(* IEC 61131-3 sources: std_i2980_v2.06_cp053/Source/IMM/ieccontrol/GlobalBaseArchives (part 14) *)

(* ---- ABMotorLockList.pu ---- *)
IMPORT_OVER_LISTFILE
 SET_ALARM
, tsListStructMotorLock
, tsDeviceId
, FBDebugTrace
, tsTraceLevel
, tsElementMotorLock
, tsSearchDataMotorLock

END_IMPORT

ALGORITHM_BLOCK ABMotorLockList #DUMMY_EDIT_BLOCK

SYSTEM_VAR
 sv_DeviceId : tsDeviceId;
 sv_TraceLevel : tsTraceLevel;
END_VAR

SYSTEM_OBJECT
 erListOverflow : ALARM;
END_OBJECT

VAR
 mListStruct : tsListStructMotorLock;
 miNextFree : DINT;
 miLowBound : DINT;
 miHighBound : DINT;
 mbInit : BOOL;
 miLastFound : DINT;
 miActElement : DINT;
 fbDebugTrace : FBDebugTrace;
END_VAR

ALGORITHM aInit

#BEGIN_EDIT_BLOCK
miLowBound := GET_LOW_BOUND(mListStruct.List);
miHighBound := GET_HIGH_BOUND(mListStruct.List);
miNextFree := miLowBound;
miLastFound := miLowBound;
miActElement := miLowBound;
mbInit := TRUE;

;#END_EDIT_BLOCK END_ALGORITHM

ALGORITHM aAdd

VAR_INPUT
 Element : tsElementMotorLock;
END_VAR
#BEGIN_EDIT_BLOCK
IF NOT mbInit THEN RETURN;; END_IF;

IF miNextFree < miHighBound THEN

    mListStruct.List[miNextFree] := Element;
    mListStruct.Used[miNextFree] := TRUE;
    miNextFree := miNextFree + 1;
ELSE
    //error: List Full
    SET_ALARM(Name := erListOverflow,
              SubID1 := sv_DeviceId.CompId,
              SubID2 := sv_DeviceId.IndexId,
              Param1 := 'ABMotorLockList.aAdd');
END_IF;

;#END_EDIT_BLOCK END_ALGORITHM

ALGORITHM aAddAt

VAR_INPUT
 Element : tsElementMotorLock;
 iPos : DINT;
END_VAR

VAR_TEMP
 i : DINT;
END_VAR

VAR
 iStart : DINT;
 iEnd : DINT;
END_VAR
#BEGIN_EDIT_BLOCK
IF NOT mbInit THEN RETURN; END_IF;

IF miNextFree <= miHighBound THEN
    IF iPos < miHighBound AND iPos >= miLowBound THEN

        IF iPos < miNextFree THEN

            iStart := miNextFree;
            iEnd := iPos+1;
        ELSE
            i := iPos;
            iEnd := miNextFree;
        END_IF;
        miNextFree := i + 1;

        //reorganize list
        FOR i := iStart TO iEnd BY -1 DO
            mListStruct.List[i] := mListStruct.List[i-1];
            mListStruct.Used[i] := TRUE;
        END_FOR;
        //adding Element
        mListStruct.List[iPos] := Element;
        mListStruct.Used[iPos] := TRUE;
    ELSE
        //error: out of bounds
        IF sv_TraceLevel.bApplication THEN
            fbDebugTrace(sText := 'ABMotorLockList.aAddAt: Error: Out of ListBounds');
        END_IF;
    END_IF;
ELSE
    //error: List Full
    SET_ALARM(Name := erListOverflow,
            SubID1 := sv_DeviceId.CompId,
            SubID2 := sv_DeviceId.IndexId,
            Param1 := 'ABMotorLockList.aAddAt');
END_IF;

;#END_EDIT_BLOCK END_ALGORITHM

ALGORITHM aSearch

VAR_INPUT
 SearchData : tsSearchDataMotorLock;
END_VAR

VAR_OUTPUT
 Element : tsElementMotorLock;
 iPos : DINT;
 bFound : BOOL;
END_VAR

VAR_TEMP
 i : DINT;
END_VAR
#BEGIN_EDIT_BLOCK
IF NOT mbInit THEN RETURN;; END_IF;

iPos := 0;
bFound := FALSE;

FOR i := miLowBound TO miNextFree-1 DO

    IF mListStruct.List[i].SearchData = SearchData THEN

       Element := mListStruct.List[i];
       //remember foundposition for aSearchNext
       miLastFound := i;
       iPos := i;
       bFound := TRUE;
       RETURN;;
    END_IF;
END_FOR;

;#END_EDIT_BLOCK END_ALGORITHM

ALGORITHM aSearchNext

VAR_INPUT
 SearchData : tsSearchDataMotorLock;
END_VAR

VAR_OUTPUT
 Element : tsElementMotorLock;
 iPos : DINT;
 bFound : BOOL;
END_VAR

VAR_TEMP
 i : DINT;
END_VAR
#BEGIN_EDIT_BLOCK
IF NOT mbInit THEN RETURN;; END_IF;

iPos := 0;
bFound := FALSE;

FOR i := miLastFound+1 TO miNextFree-1 DO

    IF mListStruct.List[i].SearchData = SearchData THEN

       Element := mListStruct.List[i];
       //remember foundposition for then next aSearchNext
       miLastFound := i;
       iPos := i;
       bFound := TRUE;
       RETURN;;
    END_IF;
END_FOR;

;#END_EDIT_BLOCK END_ALGORITHM

ALGORITHM aRemove

VAR_INPUT
 SearchData : tsSearchDataMotorLock;
END_VAR

VAR_OUTPUT
 Element : tsElementMotorLock;
 iPos : DINT;
 bFound : BOOL;
END_VAR

VAR_TEMP
 i : DINT;
END_VAR
#BEGIN_EDIT_BLOCK
IF NOT mbInit THEN RETURN; END_IF;

iPos := 0;
bFound := FALSE;

FOR i := miLowBound TO miNextFree-1 DO

    IF mListStruct.List[i].SearchData = SearchData THEN

       iPos := i;
       bFound := TRUE;
       Element := mListStruct.List[i];
       //reorganize list
       FOR i := iPos TO miNextFree-1 DO
           mListStruct.List[i] := mListStruct.List[i+1];
       END_FOR;
       mListStruct.Used[miNextFree - 1] := FALSE;
       miNextFree := miNextFree - 1;
       RETURN;
    END_IF;
END_FOR;

;#END_EDIT_BLOCK END_ALGORITHM

ALGORITHM aRemoveAt

VAR_INPUT
 iPos : DINT;
END_VAR

VAR_OUTPUT
 Element : tsElementMotorLock;
END_VAR

VAR_TEMP
 i : DINT;
END_VAR
#BEGIN_EDIT_BLOCK
IF NOT mbInit THEN RETURN; END_IF;

IF iPos <= miHighBound AND iPos >= miLowBound THEN

    Element:= mListStruct.List[iPos];
    miActElement := iPos;

    //reorganize list
    FOR i := iPos TO miNextFree-1 DO
        mListStruct.List[i] := mListStruct.List[i+1];
    END_FOR;
    mListStruct.Used[miNextFree - 1] := FALSE;

    miNextFree := miNextFree - 1;
ELSE
    //error: out of bounds
    IF sv_TraceLevel.bApplication THEN
        fbDebugTrace(sText := 'ABMotorLockList.aRemoveAt: Error: Out of ListBounds');
    END_IF;
END_IF;

;#END_EDIT_BLOCK END_ALGORITHM

ALGORITHM aRemoveAll

VAR_TEMP
 i : DINT;
END_VAR
#BEGIN_EDIT_BLOCK
IF NOT mbInit THEN RETURN; END_IF;
FOR i := miNextFree-1 TO miLowBound DO
    //clearing the whole list
    mListStruct.Used[i] := FALSE;
END_FOR;
miNextFree := miLowBound;

;#END_EDIT_BLOCK END_ALGORITHM

ALGORITHM aElementAt

VAR_OUTPUT
 Element : tsElementMotorLock;
END_VAR

VAR_INPUT
 iPos : DINT;
END_VAR
#BEGIN_EDIT_BLOCK
IF NOT mbInit THEN RETURN; END_IF;

IF iPos <= miHighBound AND iPos >= miLowBound THEN

    Element := mListStruct.List[iPos];
    miActElement := iPos;
ELSE
    //error: out of bounds
    IF sv_TraceLevel.bApplication THEN
        fbDebugTrace(sText := 'ABMotorLockList.aElementAt: Error: Out of ListBounds');
    END_IF;
END_IF;

;#END_EDIT_BLOCK END_ALGORITHM

ALGORITHM aModifyAt

VAR_INPUT
 iPos : DINT;
END_VAR

VAR_IN_OUT
 Element : tsElementMotorLock;
END_VAR
#BEGIN_EDIT_BLOCK
IF NOT mbInit THEN RETURN; END_IF;

IF iPos <= miHighBound AND iPos >= miLowBound THEN

     mListStruct.List[iPos] := Element;
     miActElement := iPos;
ELSE
    //error: out of bounds
    IF sv_TraceLevel.bApplication THEN
        fbDebugTrace(sText := 'ABMotorLockList.aModifyAt: Error: Out of ListBounds');
    END_IF;
END_IF;

;#END_EDIT_BLOCK END_ALGORITHM

// ALGORITHM aGetSize

// #BEGIN_EDIT_BLOCK
// IF NOT mbInit THEN RETURN; END_IF;
// //returns the size of the list
// iSize := miHighBound - miLowBound;

// ;#END_EDIT_BLOCK END_ALGORITHM

// ALGORITHM aGetElementsCount

// VAR_OUTPUT
 // iUsed : DINT;
// END_VAR
// #BEGIN_EDIT_BLOCK
// IF NOT mbInit THEN RETURN; END_IF;
//
// iUsed := miNextFree - miLowBound;

// ;#END_EDIT_BLOCK END_ALGORITHM

FUNCTION aGetSize : DINT
 #DUMMY_EDIT_BLOCK
#BEGIN_EDIT_BLOCK
IF NOT mbInit THEN RETURN; END_IF;
//returns the size of the list
aGetSize := miHighBound - miLowBound;

;#END_EDIT_BLOCK END_FUNCTION

FUNCTION aGetElementCount : DINT
 #DUMMY_EDIT_BLOCK
#BEGIN_EDIT_BLOCK
IF NOT mbInit THEN RETURN; END_IF;

aGetElementCount:= miNextFree - miLowBound;

;#END_EDIT_BLOCK END_FUNCTION

ALGORITHM aFirstElement

VAR_OUTPUT
 Element : tsElementMotorLock;
END_VAR
#BEGIN_EDIT_BLOCK
IF NOT mbInit THEN RETURN; END_IF;

miActElement := miLowBound;
Element := mListStruct.List[miLowBound];

;#END_EDIT_BLOCK END_ALGORITHM

ALGORITHM aNextElement

VAR_OUTPUT
 Element : tsElementMotorLock;
 iPos : DINT;
END_VAR
#BEGIN_EDIT_BLOCK
IF NOT mbInit THEN RETURN; END_IF;

IF miActElement < miHighBound THEN

    miActElement := miActElement + 1;
    iPos := miActElement;
    Element := mListStruct.List[miActElement];
END_IF;

;#END_EDIT_BLOCK END_ALGORITHM

ALGORITHM aLastElement

VAR_OUTPUT
 Element : tsElementMotorLock;
END_VAR
#BEGIN_EDIT_BLOCK
IF NOT mbInit THEN RETURN; END_IF;

miActElement := miNextFree - 1;
Element := mListStruct.List[miActElement];

;#END_EDIT_BLOCK END_ALGORITHM

ALGORITHM aPrevElement

VAR_OUTPUT
 Element : tsElementMotorLock;
 iPos : DINT;
END_VAR
#BEGIN_EDIT_BLOCK
IF NOT mbInit THEN RETURN; END_IF;

IF miActElement > miLowBound THEN

    miActElement := miActElement - 1;
    iPos := miActElement;
    Element := mListStruct.List[miActElement];
END_IF;

;#END_EDIT_BLOCK END_ALGORITHM

ALGORITHM aImport

VAR_INPUT
 ListStruct : tsListStructMotorLock;
END_VAR

VAR_TEMP
 i : DINT;
END_VAR
#BEGIN_EDIT_BLOCK
IF NOT mbInit THEN RETURN; END_IF;

miLastFound := miLowBound;
miActElement := miLowBound;
miNextFree := miLowBound;
mListStruct :=  ListStruct;

//cheching used elements
FOR i := miLowBound TO miHighBound DO

   IF NOT mListStruct.Used[i] THEN
        miNextFree := i;
        RETURN;
   END_IF;
END_FOR;

;#END_EDIT_BLOCK END_ALGORITHM

ALGORITHM aExport

VAR_OUTPUT
 ListStruct : tsListStructMotorLock;
END_VAR
#BEGIN_EDIT_BLOCK
IF NOT mbInit THEN RETURN; END_IF;

ListStruct := mListStruct;

;#END_EDIT_BLOCK END_ALGORITHM

END_ALGORITHM_BLOCK

#END_OF_IEC_PART

@Puma @IecEditor 6 68 @Pou 25
@@@BEG_Comment@@@

@@@END_Comment@@@

@BEG_Contents

@BEG_Func
@RT(17)FuncTreeContainer
1
@Var @RT(9)SET_ALARM @RT(0) @T @T @DERIVED 0 @F @RT(23)KEBA_STANDARD_PROCEDURE @F
@T
@BEG_Attrib
0 @RT(0) @RT(0)
@END_Attrib
1 1 @F @F @F @F

@END_Func

@BEG_Const
@RT(18)ConstTreeContainer
0
@END_Const

@BEG_Export

@BEG_Kind
@ALGORITHM_BLOCK @RT(15)ABMotorLockList @STRUCTURED_TEXT
@RT(0) @RT(0) @RT(0)
@END_Kind

@BEG_Dcl
@RT(16)DclTreeContainer
11
@Var @RT(14)erListOverflow @RT(0) @T @F @DT @RT(5)ALARM @RT(0) @T @T @BASIC 0 @F
@F @F
@T
@BEG_Attrib
3 @RT(0) @RT(0) @RT(0)
@END_Attrib
1 7 @F @F @F @F

@Var @RT(11)mListStruct @RT(0) @T @T @DERIVED 0 @T @T @DT @RT(21)tsListStructMotorLock @RT(0) @T @T @UNKNOWN 0 @F
@F @F
@T
@BEG_Attrib
3 @RT(0) @RT(0) @RT(0)
@END_Attrib
1 0 @F @F @F @F

@Var @RT(10)miNextFree @RT(0) @T @F @DT @RT(4)DINT @RT(0) @T @T @BASIC 0 @F
@F @F
@T
@BEG_Attrib
3 @RT(0) @RT(0) @RT(0)
@END_Attrib
1 0 @F @F @F @F

@Var @RT(10)miLowBound @RT(0) @T @F @DT @RT(4)DINT @RT(0) @T @T @BASIC 0 @F
@F @F
@T
@BEG_Attrib
3 @RT(0) @RT(0) @RT(0)
@END_Attrib
1 0 @F @F @F @F

@Var @RT(11)miHighBound @RT(0) @T @F @DT @RT(4)DINT @RT(0) @T @T @BASIC 0 @F
@F @F
@T
@BEG_Attrib
3 @RT(0) @RT(0) @RT(0)
@END_Attrib
1 0 @F @F @F @F

@Var @RT(6)mbInit @RT(0) @T @F @DT @RT(4)BOOL @RT(0) @T @T @BASIC 0 @F
@F @F
@T
@BEG_Attrib
3 @RT(0) @RT(0) @RT(0)
@END_Attrib
1 0 @F @F @F @F

@Var @RT(11)miLastFound @RT(0) @T @F @DT @RT(4)DINT @RT(0) @T @T @BASIC 0 @F
@F @F
@T
@BEG_Attrib
3 @RT(0) @RT(0) @RT(0)
@END_Attrib
1 0 @F @F @F @F

@Var @RT(12)miActElement @RT(0) @T @F @DT @RT(4)DINT @RT(0) @T @T @BASIC 0 @F
@F @F
@T
@BEG_Attrib
3 @RT(0) @RT(0) @RT(0)
@END_Attrib
1 0 @F @F @F @F

@Var @RT(11)sv_DeviceId @RT(0) @T @T @DERIVED 0 @T @T @DT @RT(10)tsDeviceId @RT(0) @T @T @UNKNOWN 0 @F
@F @F
@T
@BEG_Attrib
3 @RT(0) @RT(0) @RT(0)
@END_Attrib
1 8 @F @F @F @F

@Var @RT(12)fbDebugTrace @RT(0) @T @T @DERIVED 0 @T @T @DT @RT(12)FBDebugTrace @RT(0) @T @T @UNKNOWN 0 @F
@F @F
@T
@BEG_Attrib
3 @RT(0) @RT(0) @RT(0)
@END_Attrib
1 0 @F @F @F @F

@Var @RT(13)sv_TraceLevel @RT(0) @T @T @DERIVED 0 @T @T @DT @RT(12)tsTraceLevel @RT(0) @T @T @UNKNOWN 0 @F
@F @F
@T
@BEG_Attrib
3 @RT(0) @RT(0) @RT(0)
@END_Attrib
1 8 @F @F @F @F

@END_Dcl

@END_Export

@BEG_Body

20

@BEG_Export

@BEG_Algo
@ALGORITHM @RT(5)aInit @STRUCTURED_TEXT
@RT(0) @RT(0) @RT(0) @F @F
@END_Algo

@BEG_Dcl
@RT(16)DclTreeContainer
0
@END_Dcl

@END_Export

@BEG_Export

@BEG_Algo
@ALGORITHM @RT(4)aAdd @STRUCTURED_TEXT
@RT(0) @RT(0) @RT(0) @F @F
@END_Algo

@BEG_Dcl
@RT(16)DclTreeContainer
1
@Var @RT(7)Element @RT(0) @T @T @DERIVED 0 @T @T @DT @RT(18)tsElementMotorLock @RT(0) @T @T @UNKNOWN 0 @F
@F @F
@T
@BEG_Attrib
3 @RT(0) @RT(0) @RT(0)
@END_Attrib
1 1 @F @F @F @F

@END_Dcl

@END_Export

@BEG_Export

@BEG_Algo
@ALGORITHM @RT(6)aAddAt @STRUCTURED_TEXT
@RT(0) @RT(0) @RT(0) @F @F
@END_Algo

@BEG_Dcl
@RT(16)DclTreeContainer
5
@Var @RT(7)Element @RT(0) @T @T @DERIVED 0 @T @T @DT @RT(18)tsElementMotorLock @RT(0) @T @T @UNKNOWN 0 @F
@F @F
@T
@BEG_Attrib
3 @RT(0) @RT(0) @RT(0)
@END_Attrib
1 1 @F @F @F @F

@Var @RT(4)iPos @RT(0) @T @F @DT @RT(4)DINT @RT(0) @T @T @BASIC 0 @F
@F @F
@T
@BEG_Attrib
3 @RT(0) @RT(0) @RT(0)
@END_Attrib
1 1 @F @F @F @F

@Var @RT(1)i @RT(0) @T @F @DT @RT(4)DINT @RT(0) @T @T @BASIC 0 @F
@F @F
@T
@BEG_Attrib
3 @RT(0) @RT(0) @RT(0)
@END_Attrib
1 4 @F @F @F @F

@Var @RT(6)iStart @RT(0) @T @F @DT @RT(4)DINT @RT(0) @T @T @BASIC 0 @F
@F @F
@T
@BEG_Attrib
3 @RT(0) @RT(0) @RT(0)
@END_Attrib
1 0 @F @F @F @F

@Var @RT(4)iEnd @RT(0) @T @F @DT @RT(4)DINT @RT(0) @T @T @BASIC 0 @F
@F @F
@T
@BEG_Attrib
3 @RT(0) @RT(0) @RT(0)
@END_Attrib
1 0 @F @F @F @F

@END_Dcl

@END_Export

@BEG_Export

@BEG_Algo
@ALGORITHM @RT(7)aSearch @STRUCTURED_TEXT
@RT(0) @RT(0) @RT(0) @F @F
@END_Algo

@BEG_Dcl
@RT(16)DclTreeContainer
5
@Var @RT(10)SearchData @RT(0) @T @T @DERIVED 0 @T @T @DT @RT(21)tsSearchDataMotorLock @RT(0) @T @T @UNKNOWN 0 @F
@F @F
@T
@BEG_Attrib
3 @RT(0) @RT(0) @RT(0)
@END_Attrib
1 1 @F @F @F @F

@Var @RT(7)Element @RT(0) @T @T @DERIVED 0 @T @T @DT @RT(18)tsElementMotorLock @RT(0) @T @T @UNKNOWN 0 @F
@F @F
@T
@BEG_Attrib
3 @RT(0) @RT(0) @RT(0)
@END_Attrib
1 3 @F @F @F @F

@Var @RT(4)iPos @RT(0) @T @F @DT @RT(4)DINT @RT(0) @T @T @BASIC 0 @F
@F @F
@T
@BEG_Attrib
3 @RT(0) @RT(0) @RT(0)
@END_Attrib
1 3 @F @F @F @F

@Var @RT(6)bFound @RT(0) @T @F @DT @RT(4)BOOL @RT(0) @T @T @BASIC 0 @F
@F @F
@T
@BEG_Attrib
3 @RT(0) @RT(0) @RT(0)
@END_Attrib
1 3 @F @F @F @F

@Var @RT(1)i @RT(0) @T @F @DT @RT(4)DINT @RT(0) @T @T @BASIC 0 @F
@F @F
@T
@BEG_Attrib
3 @RT(0) @RT(0) @RT(0)
@END_Attrib
1 4 @F @F @F @F

@END_Dcl

@END_Export

@BEG_Export

@BEG_Algo
@ALGORITHM @RT(11)aSearchNext @STRUCTURED_TEXT
@RT(0) @RT(0) @RT(0) @F @F
@END_Algo

@BEG_Dcl
@RT(16)DclTreeContainer
5
@Var @RT(10)SearchData @RT(0) @T @T @DERIVED 0 @T @T @DT @RT(21)tsSearchDataMotorLock @RT(0) @T @T @UNKNOWN 0 @F
@F @F
@T
@BEG_Attrib
3 @RT(0) @RT(0) @RT(0)
@END_Attrib
1 1 @F @F @F @F

@Var @RT(7)Element @RT(0) @T @T @DERIVED 0 @T @T @DT @RT(18)tsElementMotorLock @RT(0) @T @T @UNKNOWN 0 @F
@F @F
@T
@BEG_Attrib
3 @RT(0) @RT(0) @RT(0)
@END_Attrib
1 3 @F @F @F @F

@Var @RT(4)iPos @RT(0) @T @F @DT @RT(4)DINT @RT(0) @T @T @BASIC 0 @F
@F @F
@T
@BEG_Attrib
3 @RT(0) @RT(0) @RT(0)
@END_Attrib
1 3 @F @F @F @F

@Var @RT(6)bFound @RT(0) @T @F @DT @RT(4)BOOL @RT(0) @T @T @BASIC 0 @F
@F @F
@T
@BEG_Attrib
3 @RT(0) @RT(0) @RT(0)
@END_Attrib
1 3 @F @F @F @F

@Var @RT(1)i @RT(0) @T @F @DT @RT(4)DINT @RT(0) @T @T @BASIC 0 @F
@F @F
@T
@BEG_Attrib
3 @RT(0) @RT(0) @RT(0)
@END_Attrib
1 4 @F @F @F @F

@END_Dcl

@END_Export

@BEG_Export

@BEG_Algo
@ALGORITHM @RT(7)aRemove @STRUCTURED_TEXT
@RT(0) @RT(0) @RT(0) @F @F
@END_Algo

@BEG_Dcl
@RT(16)DclTreeContainer
5
@Var @RT(10)SearchData @RT(0) @T @T @DERIVED 0 @T @T @DT @RT(21)tsSearchDataMotorLock @RT(0) @T @T @UNKNOWN 0 @F
@F @F
@T
@BEG_Attrib
3 @RT(0) @RT(0) @RT(0)
@END_Attrib
1 1 @F @F @F @F

@Var @RT(7)Element @RT(0) @T @T @DERIVED 0 @T @T @DT @RT(18)tsElementMotorLock @RT(0) @T @T @UNKNOWN 0 @F
@F @F
@T
@BEG_Attrib
3 @RT(0) @RT(0) @RT(0)
@END_Attrib
1 3 @F @F @F @F

@Var @RT(4)iPos @RT(0) @T @F @DT @RT(4)DINT @RT(0) @T @T @BASIC 0 @F
@F @F
@T
@BEG_Attrib
3 @RT(0) @RT(0) @RT(0)
@END_Attrib
1 3 @F @F @F @F

@Var @RT(6)bFound @RT(0) @T @F @DT @RT(4)BOOL @RT(0) @T @T @BASIC 0 @F
@F @F
@T
@BEG_Attrib
3 @RT(0) @RT(0) @RT(0)
@END_Attrib
1 3 @F @F @F @F

@Var @RT(1)i @RT(0) @T @F @DT @RT(4)DINT @RT(0) @T @T @BASIC 0 @F
@F @F
@T
@BEG_Attrib
3 @RT(0) @RT(0) @RT(0)
@END_Attrib
1 4 @F @F @F @F

@END_Dcl

@END_Export

@BEG_Export

@BEG_Algo
@ALGORITHM @RT(9)aRemoveAt @STRUCTURED_TEXT
@RT(0) @RT(0) @RT(0) @F @F
@END_Algo

@BEG_Dcl
@RT(16)DclTreeContainer
3
@Var @RT(4)iPos @RT(0) @T @F @DT @RT(4)DINT @RT(0) @T @T @BASIC 0 @F
@F @F
@T
@BEG_Attrib
3 @RT(0) @RT(0) @RT(0)
@END_Attrib
1 1 @F @F @F @F

@Var @RT(7)Element @RT(0) @T @T @DERIVED 0 @T @T @DT @RT(18)tsElementMotorLock @RT(0) @T @T @UNKNOWN 0 @F
@F @F
@T
@BEG_Attrib
3 @RT(0) @RT(0) @RT(0)
@END_Attrib
1 3 @F @F @F @F

@Var @RT(1)i @RT(0) @T @F @DT @RT(4)DINT @RT(0) @T @T @BASIC 0 @F
@F @F
@T
@BEG_Attrib
3 @RT(0) @RT(0) @RT(0)
@END_Attrib
1 4 @F @F @F @F

@END_Dcl

@END_Export

@BEG_Export

@BEG_Algo
@ALGORITHM @RT(10)aRemoveAll @STRUCTURED_TEXT
@RT(0) @RT(0) @RT(0) @F @F
@END_Algo

@BEG_Dcl
@RT(16)DclTreeContainer
1
@Var @RT(1)i @RT(0) @T @F @DT @RT(4)DINT @RT(0) @T @T @BASIC 0 @F
@F @F
@T
@BEG_Attrib
3 @RT(0) @RT(0) @RT(0)
@END_Attrib
1 4 @F @F @F @F

@END_Dcl

@END_Export

@BEG_Export

@BEG_Algo
@ALGORITHM @RT(10)aElementAt @STRUCTURED_TEXT
@RT(0) @RT(0) @RT(0) @F @F
@END_Algo

@BEG_Dcl
@RT(16)DclTreeContainer
2
@Var @RT(7)Element @RT(0) @T @T @DERIVED 0 @T @T @DT @RT(18)tsElementMotorLock @RT(0) @T @T @UNKNOWN 0 @F
@F @F
@T
@BEG_Attrib
3 @RT(0) @RT(0) @RT(0)
@END_Attrib
1 3 @F @F @F @F

@Var @RT(4)iPos @RT(0) @T @F @DT @RT(4)DINT @RT(0) @T @T @BASIC 0 @F
@F @F
@T
@BEG_Attrib
3 @RT(0) @RT(0) @RT(0)
@END_Attrib
1 1 @F @F @F @F

@END_Dcl

@END_Export

@BEG_Export

@BEG_Algo
@ALGORITHM @RT(9)aModifyAt @STRUCTURED_TEXT
@RT(0) @RT(0) @RT(0) @F @F
@END_Algo

@BEG_Dcl
@RT(16)DclTreeContainer
2
@Var @RT(4)iPos @RT(0) @T @F @DT @RT(4)DINT @RT(0) @T @T @BASIC 0 @F
@F @F
@T
@BEG_Attrib
3 @RT(0) @RT(0) @RT(0)
@END_Attrib
1 1 @F @F @F @F

@Var @RT(7)Element @RT(0) @T @T @DERIVED 0 @T @T @DT @RT(18)tsElementMotorLock @RT(0) @T @T @UNKNOWN 0 @F
@F @F
@T
@BEG_Attrib
3 @RT(0) @RT(0) @RT(0)
@END_Attrib
1 2 @F @F @F @F

@END_Dcl

@END_Export

@BEG_Export

@BEG_Algo
@ALGORITHM @RT(8)aGetSize @STRUCTURED_TEXT
@RT(0) @RT(0) @RT(0) @F @T
@END_Algo

@BEG_Dcl
@RT(16)DclTreeContainer
0
@END_Dcl

@END_Export

@BEG_Export

@BEG_Algo
@ALGORITHM @RT(17)aGetElementsCount @STRUCTURED_TEXT
@RT(0) @RT(0) @RT(0) @F @T
@END_Algo

@BEG_Dcl
@RT(16)DclTreeContainer
1
@Var @RT(5)iUsed @RT(0) @T @F @DT @RT(4)DINT @RT(0) @T @T @BASIC 0 @F
@F @F
@T
@BEG_Attrib
3 @RT(0) @RT(0) @RT(0)
@END_Attrib
1 3 @F @F @F @F

@END_Dcl

@END_Export

@BEG_Export

@BEG_Algo
@FUNCTION @RT(8)aGetSize @STRUCTURED_TEXT
@RT(4)DINT @RT(0) @RT(0) @F @F
@END_Algo

@BEG_Dcl
@RT(16)DclTreeContainer
0
@END_Dcl

@END_Export

@BEG_Export

@BEG_Algo
@FUNCTION @RT(16)aGetElementCount @STRUCTURED_TEXT
@RT(4)DINT @RT(0) @RT(0) @F @F
@END_Algo

@BEG_Dcl
@RT(16)DclTreeContainer
0
@END_Dcl

@END_Export

@BEG_Export

@BEG_Algo
@ALGORITHM @RT(13)aFirstElement @STRUCTURED_TEXT
@RT(0) @RT(0) @RT(0) @F @F
@END_Algo

@BEG_Dcl
@RT(16)DclTreeContainer
1
@Var @RT(7)Element @RT(0) @T @T @DERIVED 0 @T @T @DT @RT(18)tsElementMotorLock @RT(0) @T @T @UNKNOWN 0 @F
@F @F
@T
@BEG_Attrib
3 @RT(0) @RT(0) @RT(0)
@END_Attrib
1 3 @F @F @F @F

@END_Dcl

@END_Export

@BEG_Export

@BEG_Algo
@ALGORITHM @RT(12)aNextElement @STRUCTURED_TEXT
@RT(0) @RT(0) @RT(0) @F @F
@END_Algo

@BEG_Dcl
@RT(16)DclTreeContainer
2
@Var @RT(7)Element @RT(0) @T @T @DERIVED 0 @T @T @DT @RT(18)tsElementMotorLock @RT(0) @T @T @UNKNOWN 0 @F
@F @F
@T
@BEG_Attrib
3 @RT(0) @RT(0) @RT(0)
@END_Attrib
1 3 @F @F @F @F

@Var @RT(4)iPos @RT(0) @T @F @DT @RT(4)DINT @RT(0) @T @T @BASIC 0 @F
@F @F
@T
@BEG_Attrib
3 @RT(0) @RT(0) @RT(0)
@END_Attrib
1 3 @F @F @F @F

@END_Dcl

@END_Export

@BEG_Export

@BEG_Algo
@ALGORITHM @RT(12)aLastElement @STRUCTURED_TEXT
@RT(0) @RT(0) @RT(0) @F @F
@END_Algo

@BEG_Dcl
@RT(16)DclTreeContainer
1
@Var @RT(7)Element @RT(0) @T @T @DERIVED 0 @T @T @DT @RT(18)tsElementMotorLock @RT(0) @T @T @UNKNOWN 0 @F
@F @F
@T
@BEG_Attrib
3 @RT(0) @RT(0) @RT(0)
@END_Attrib
1 3 @F @F @F @F

@END_Dcl

@END_Export

@BEG_Export

@BEG_Algo
@ALGORITHM @RT(12)aPrevElement @STRUCTURED_TEXT
@RT(0) @RT(0) @RT(0) @F @F
@END_Algo

@BEG_Dcl
@RT(16)DclTreeContainer
2
@Var @RT(7)Element @RT(0) @T @T @DERIVED 0 @T @T @DT @RT(18)tsElementMotorLock @RT(0) @T @T @UNKNOWN 0 @F
@F @F
@T
@BEG_Attrib
3 @RT(0) @RT(0) @RT(0)
@END_Attrib
1 3 @F @F @F @F

@Var @RT(4)iPos @RT(0) @T @F @DT @RT(4)DINT @RT(0) @T @T @BASIC 0 @F
@F @F
@T
@BEG_Attrib
3 @RT(0) @RT(0) @RT(0)
@END_Attrib
1 3 @F @F @F @F

@END_Dcl

@END_Export

@BEG_Export

@BEG_Algo
@ALGORITHM @RT(7)aImport @STRUCTURED_TEXT
@RT(0) @RT(0) @RT(0) @F @F
@END_Algo

@BEG_Dcl
@RT(16)DclTreeContainer
2
@Var @RT(10)ListStruct @RT(0) @T @T @DERIVED 0 @T @T @DT @RT(21)tsListStructMotorLock @RT(0) @T @T @UNKNOWN 0 @F
@F @F
@T
@BEG_Attrib
3 @RT(0) @RT(0) @RT(0)
@END_Attrib
1 1 @F @F @F @F

@Var @RT(1)i @RT(0) @T @F @DT @RT(4)DINT @RT(0) @T @T @BASIC 0 @F
@F @F
@T
@BEG_Attrib
3 @RT(0) @RT(0) @RT(0)
@END_Attrib
1 4 @F @F @F @F

@END_Dcl

@END_Export

@BEG_Export

@BEG_Algo
@ALGORITHM @RT(7)aExport @STRUCTURED_TEXT
@RT(0) @RT(0) @RT(0) @F @F
@END_Algo

@BEG_Dcl
@RT(16)DclTreeContainer
1
@Var @RT(10)ListStruct @RT(0) @T @T @DERIVED 0 @T @T @DT @RT(21)tsListStructMotorLock @RT(0) @T @T @UNKNOWN 0 @F
@F @F
@T
@BEG_Attrib
3 @RT(0) @RT(0) @RT(0)
@END_Attrib
1 3 @F @F @F @F

@END_Dcl

@END_Export

@BEG_Body
@TL(7)
miLowBound := GET_LOW_BOUND(mListStruct.List);
miHighBound := GET_HIGH_BOUND(mListStruct.List);
miNextFree := miLowBound;
miLastFound := miLowBound;
miActElement := miLowBound;
mbInit := TRUE;

@END_Body

@@@BEG_Comment@@@
@TL(0)

@@@END_Comment@@@

@BEG_Body
@TL(15)
IF NOT mbInit THEN RETURN;; END_IF;

IF miNextFree < miHighBound THEN

    mListStruct.List[miNextFree] := Element;
    mListStruct.Used[miNextFree] := TRUE;
    miNextFree := miNextFree + 1;
ELSE
    //error: List Full
    SET_ALARM(Name := erListOverflow,
              SubID1 := sv_DeviceId.CompId,
              SubID2 := sv_DeviceId.IndexId,
              Param1 := 'ABMotorLockList.aAdd');
END_IF;

@END_Body

@@@BEG_Comment@@@
@TL(0)

@@@END_Comment@@@

@BEG_Body
@TL(37)
IF NOT mbInit THEN RETURN; END_IF;

IF miNextFree <= miHighBound THEN
    IF iPos < miHighBound AND iPos >= miLowBound THEN

        IF iPos < miNextFree THEN

            iStart := miNextFree;
            iEnd := iPos+1;
        ELSE
            i := iPos;
            iEnd := miNextFree;
        END_IF;
        miNextFree := i + 1;

        //reorganize list
        FOR i := iStart TO iEnd BY -1 DO
            mListStruct.List[i] := mListStruct.List[i-1];
            mListStruct.Used[i] := TRUE;
        END_FOR;
        //adding Element
        mListStruct.List[iPos] := Element;
        mListStruct.Used[iPos] := TRUE;
    ELSE
        //error: out of bounds
        IF sv_TraceLevel.bApplication THEN
            fbDebugTrace(sText := 'ABMotorLockList.aAddAt: Error: Out of ListBounds');
        END_IF;
    END_IF;
ELSE
    //error: List Full
    SET_ALARM(Name := erListOverflow,
            SubID1 := sv_DeviceId.CompId,
            SubID2 := sv_DeviceId.IndexId,
            Param1 := 'ABMotorLockList.aAddAt');
END_IF;

@END_Body

@@@BEG_Comment@@@
@TL(0)

@@@END_Comment@@@

@BEG_Body
@TL(18)
IF NOT mbInit THEN RETURN;; END_IF;

iPos := 0;
bFound := FALSE;

FOR i := miLowBound TO miNextFree-1 DO

    IF mListStruct.List[i].SearchData = SearchData THEN

       Element := mListStruct.List[i];
       //remember foundposition for aSearchNext
       miLastFound := i;
       iPos := i;
       bFound := TRUE;
       RETURN;;
    END_IF;
END_FOR;

@END_Body

@@@BEG_Comment@@@
@TL(0)

@@@END_Comment@@@

@BEG_Body
@TL(19)
IF NOT mbInit THEN RETURN;; END_IF;

iPos := 0;
bFound := FALSE;

FOR i := miLastFound+1 TO miNextFree-1 DO

    IF mListStruct.List[i].SearchData = SearchData THEN

       Element := mListStruct.List[i];
       //remember foundposition for then next aSearchNext
       miLastFound := i;
       iPos := i;
       bFound := TRUE;
       RETURN;;
    END_IF;
END_FOR;

@END_Body

@@@BEG_Comment@@@
@TL(0)

@@@END_Comment@@@

@BEG_Body
@TL(22)
IF NOT mbInit THEN RETURN; END_IF;

iPos := 0;
bFound := FALSE;

FOR i := miLowBound TO miNextFree-1 DO

    IF mListStruct.List[i].SearchData = SearchData THEN

       iPos := i;
       bFound := TRUE;
       Element := mListStruct.List[i];
       //reorganize list
       FOR i := iPos TO miNextFree-1 DO
           mListStruct.List[i] := mListStruct.List[i+1];
       END_FOR;
       mListStruct.Used[miNextFree - 1] := FALSE;
       miNextFree := miNextFree - 1;
       RETURN;
    END_IF;
END_FOR;

@END_Body

@@@BEG_Comment@@@
@TL(0)

@@@END_Comment@@@

@BEG_Body
@TL(21)
IF NOT mbInit THEN RETURN; END_IF;

IF iPos <= miHighBound AND iPos >= miLowBound THEN

    Element:= mListStruct.List[iPos];
    miActElement := iPos;

    //reorganize list
    FOR i := iPos TO miNextFree-1 DO
        mListStruct.List[i] := mListStruct.List[i+1];
    END_FOR;
    mListStruct.Used[miNextFree - 1] := FALSE;

    miNextFree := miNextFree - 1;
ELSE
    //error: out of bounds
    IF sv_TraceLevel.bApplication THEN
        fbDebugTrace(sText := 'ABMotorLockList.aRemoveAt: Error: Out of ListBounds');
    END_IF;
END_IF;

@END_Body

@@@BEG_Comment@@@
@TL(0)

@@@END_Comment@@@

@BEG_Body
@TL(7)
IF NOT mbInit THEN RETURN; END_IF;
FOR i := miNextFree-1 TO miLowBound DO
    //clearing the whole list
    mListStruct.Used[i] := FALSE;
END_FOR;
miNextFree := miLowBound;

@END_Body

@@@BEG_Comment@@@
@TL(0)

@@@END_Comment@@@

@BEG_Body
@TL(13)
IF NOT mbInit THEN RETURN; END_IF;

IF iPos <= miHighBound AND iPos >= miLowBound THEN

    Element := mListStruct.List[iPos];
    miActElement := iPos;
ELSE
    //error: out of bounds
    IF sv_TraceLevel.bApplication THEN
        fbDebugTrace(sText := 'ABMotorLockList.aElementAt: Error: Out of ListBounds');
    END_IF;
END_IF;

@END_Body

@@@BEG_Comment@@@
@TL(0)

@@@END_Comment@@@

@BEG_Body
@TL(13)
IF NOT mbInit THEN RETURN; END_IF;

IF iPos <= miHighBound AND iPos >= miLowBound THEN

     mListStruct.List[iPos] := Element;
     miActElement := iPos;
ELSE
    //error: out of bounds
    IF sv_TraceLevel.bApplication THEN
        fbDebugTrace(sText := 'ABMotorLockList.aModifyAt: Error: Out of ListBounds');
    END_IF;
END_IF;

@END_Body

@@@BEG_Comment@@@
@TL(0)

@@@END_Comment@@@

@BEG_Body
@TL(4)
IF NOT mbInit THEN RETURN; END_IF;
//returns the size of the list
iSize := miHighBound - miLowBound;

@END_Body

@@@BEG_Comment@@@
@TL(0)

@@@END_Comment@@@

@BEG_Body
@TL(4)
IF NOT mbInit THEN RETURN; END_IF;

iUsed := miNextFree - miLowBound;

@END_Body

@@@BEG_Comment@@@
@TL(0)

@@@END_Comment@@@

@BEG_Body
@TL(5)
IF NOT mbInit THEN RETURN; END_IF;
//returns the size of the list
aGetSize := miHighBound - miLowBound;

@END_Body

@@@BEG_Comment@@@
@TL(0)

@@@END_Comment@@@

@BEG_Body
@TL(5)
IF NOT mbInit THEN RETURN; END_IF;

aGetElementCount:= miNextFree - miLowBound;

@END_Body

@@@BEG_Comment@@@
@TL(0)

@@@END_Comment@@@

@BEG_Body
@TL(6)
IF NOT mbInit THEN RETURN; END_IF;

miActElement := miLowBound;
Element := mListStruct.List[miLowBound];

@END_Body

@@@BEG_Comment@@@
@TL(0)

@@@END_Comment@@@

@BEG_Body
@TL(9)
IF NOT mbInit THEN RETURN; END_IF;

IF miActElement < miHighBound THEN

    miActElement := miActElement + 1;
    iPos := miActElement;
    Element := mListStruct.List[miActElement];
END_IF;

@END_Body

@@@BEG_Comment@@@
@TL(0)

@@@END_Comment@@@

@BEG_Body
@TL(6)
IF NOT mbInit THEN RETURN; END_IF;

miActElement := miNextFree - 1;
Element := mListStruct.List[miActElement];

@END_Body

@@@BEG_Comment@@@
@TL(0)

@@@END_Comment@@@

@BEG_Body
@TL(9)
IF NOT mbInit THEN RETURN; END_IF;

IF miActElement > miLowBound THEN

    miActElement := miActElement - 1;
    iPos := miActElement;
    Element := mListStruct.List[miActElement];
END_IF;

@END_Body

@@@BEG_Comment@@@
@TL(0)

@@@END_Comment@@@

@BEG_Body
@TL(16)
IF NOT mbInit THEN RETURN; END_IF;

miLastFound := miLowBound;
miActElement := miLowBound;
miNextFree := miLowBound;
mListStruct :=  ListStruct;

//cheching used elements
FOR i := miLowBound TO miHighBound DO

   IF NOT mListStruct.Used[i] THEN
        miNextFree := i;
        RETURN;
   END_IF;
END_FOR;

@END_Body

@@@BEG_Comment@@@
@TL(0)

@@@END_Comment@@@

@BEG_Body
@TL(4)
IF NOT mbInit THEN RETURN; END_IF;

ListStruct := mListStruct;

@END_Body

@@@BEG_Comment@@@
@TL(0)

@@@END_Comment@@@
@END_Body

@END_Contents

(* ---- ABMotorLockRelease.pu ---- *)
IMPORT_OVER_LISTFILE
 ALARM_EVENT
, tsTraceLevel
, ABMotorLockList
, FBDebugTrace
, ALARM_EVENT_DATA
, tsElementMotorLock

END_IMPORT

ALGORITHM_BLOCK ABMotorLockRelease #DUMMY_EDIT_BLOCK

SYSTEM_VAR
 sv_bMotorLocked : BOOL;
 sv_TraceLevel : tsTraceLevel;
END_VAR

SYSTEM_OBJECT
 EV_Task_3 : TASK;
 evAlarmMotorLock : ALARM_EVENT;
 evAlarmMotorRelease : ALARM_EVENT;
END_OBJECT

VAR
 abMotorLockList : ABMotorLockList;
 mbInitDone : BOOL;
 miEntries : DINT;
 fbDebugTrace : FBDebugTrace;
END_VAR

EVENT_ALGORITHM evaAlarmMotorLock ON EV_Task_3 WITH evAlarmMotorLock

VAR_INPUT
 evAlarmMotorLockData : ALARM_EVENT_DATA;
END_VAR

VAR
 ElementMotorLock : tsElementMotorLock;
END_VAR
#BEGIN_EDIT_BLOCK
IF NOT mbInitDone THEN
    abMotorLockList.aInit();
    mbInitDone := TRUE;
END_IF;

IF sv_TraceLevel.bLockUnlock THEN
   fbDebugTrace(CONCAT('motor locked   by alarm ', GET_ALARM_NAME(evAlarmMotorLockData.NAME)));
END_IF;

//search if entry already exists
ElementMotorLock.SearchData.Alarm := evAlarmMotorLockData.NAME;
ElementMotorLock.SearchData.SubID1 := evAlarmMotorLockData.SUBID1;
ElementMotorLock.SearchData.SubID2 := evAlarmMotorLockData.SUBID2;
ElementMotorLock.SearchData.SubID3 := evAlarmMotorLockData.SUBID3;
ElementMotorLock.SearchData.SubID4 := evAlarmMotorLockData.SUBID4;

abMotorLockList.aSearch(SearchData := ElementMotorLock.SearchData);

IF NOT abMotorLockList.aSearch.bFound THEN
    //add entry
    ElementMotorLock.ElementData.Alarm := evAlarmMotorLockData.NAME;
    ElementMotorLock.ElementData.SubID1 := evAlarmMotorLockData.SUBID1;
    ElementMotorLock.ElementData.SubID2 := evAlarmMotorLockData.SUBID2;
    ElementMotorLock.ElementData.SubID3 := evAlarmMotorLockData.SUBID3;
    ElementMotorLock.ElementData.SubID4 := evAlarmMotorLockData.SUBID4;
    abMotorLockList.aAdd(Element := ElementMotorLock);
END_IF;

//get number of elements
miEntries := abMotorLockList.aGetElementCount();
IF miEntries > 0 THEN
    //one or more entries in the list -> release motor
    sv_bMotorLocked := TRUE;
END_IF;

;#END_EDIT_BLOCK END_ALGORITHM

EVENT_ALGORITHM evaAlarmMotorRelease ON EV_Task_3 WITH evAlarmMotorRelease

VAR_INPUT
 evAlarmMotorReleaseData : ALARM_EVENT_DATA;
END_VAR

VAR
 ElementMotorRelease : tsElementMotorLock;
END_VAR
#BEGIN_EDIT_BLOCK
IF NOT mbInitDone THEN
    abMotorLockList.aInit();
    mbInitDone := TRUE;
END_IF;

IF sv_TraceLevel.bLockUnlock THEN
   fbDebugTrace(CONCAT('motor unlocked by alarm ', GET_ALARM_NAME(evAlarmMotorReleaseData.NAME)));
END_IF;

//search if entry already exists
ElementMotorRelease.SearchData.Alarm := evAlarmMotorReleaseData.NAME;
ElementMotorRelease.SearchData.SubID1 := evAlarmMotorReleaseData.SUBID1;
ElementMotorRelease.SearchData.SubID2 := evAlarmMotorReleaseData.SUBID2;
ElementMotorRelease.SearchData.SubID3 := evAlarmMotorReleaseData.SUBID3;
ElementMotorRelease.SearchData.SubID4 := evAlarmMotorReleaseData.SUBID4;

abMotorLockList.aSearch(SearchData := ElementMotorRelease.SearchData);

IF abMotorLockList.aSearch.bFound THEN
    //remove entry
    abMotorLockList.aRemove(SearchData := ElementMotorRelease.SearchData);
END_IF;

//get number of elements
miEntries := abMotorLockList.aGetElementCount();
IF miEntries = 0 THEN
    //no lock entries left -> release motor
    sv_bMotorLocked := FALSE;
END_IF;

;#END_EDIT_BLOCK END_ALGORITHM

END_ALGORITHM_BLOCK

#END_OF_IEC_PART

@Puma @IecEditor 6 52 @Pou 25
@@@BEG_Comment@@@

@@@END_Comment@@@

@BEG_Contents

@BEG_Func
@RT(17)FuncTreeContainer
0
@END_Func

@BEG_Const
@RT(18)ConstTreeContainer
0
@END_Const

@BEG_Export

@BEG_Kind
@ALGORITHM_BLOCK @RT(18)ABMotorLockRelease @STRUCTURED_TEXT
@RT(0) @RT(0) @RT(0)
@END_Kind

@BEG_Dcl
@RT(16)DclTreeContainer
9
@Var @RT(9)EV_Task_3 @RT(0) @T @T @RENAMED 0 @T @T @DT @RT(4)TASK @RT(0) @T @T @BASIC 0 @F
@F @F
@T
@BEG_Attrib
3 @RT(0) @RT(0) @RT(0)
@END_Attrib
1 7 @F @F @F @F

@Var @RT(16)evAlarmMotorLock @RT(0) @T @T @RENAMED 0 @T @T @DT @RT(11)ALARM_EVENT @RT(0) @T @T @UNKNOWN 0 @F
@F @F
@T
@BEG_Attrib
3 @RT(0) @RT(0) @RT(0)
@END_Attrib
1 7 @F @F @F @F

@Var @RT(19)evAlarmMotorRelease @RT(0) @T @T @RENAMED 0 @T @T @DT @RT(11)ALARM_EVENT @RT(0) @T @T @UNKNOWN 0 @F
@F @F
@T
@BEG_Attrib
3 @RT(0) @RT(0) @RT(0)
@END_Attrib
1 7 @F @F @F @F

@Var @RT(15)sv_bMotorLocked @RT(0) @T @F @DT @RT(4)BOOL @RT(0) @T @T @BASIC 0 @F
@F @F
@T
@BEG_Attrib
3 @RT(0) @RT(0) @RT(0)
@END_Attrib
1 8 @F @F @F @F

@Var @RT(13)sv_TraceLevel @RT(0) @T @T @RENAMED 0 @T @T @DT @RT(12)tsTraceLevel @RT(0) @T @T @UNKNOWN 0 @F
@F @F
@T
@BEG_Attrib
3 @RT(0) @RT(0) @RT(0)
@END_Attrib
1 8 @F @F @F @F

@Var @RT(15)abMotorLockList @RT(0) @T @T @DERIVED 0 @T @T @DT @RT(15)ABMotorLockList @RT(0) @T @T @UNKNOWN 0 @F
@F @F
@T
@BEG_Attrib
3 @RT(0) @RT(0) @RT(0)
@END_Attrib
1 0 @F @F @F @F

@Var @RT(10)mbInitDone @RT(0) @T @F @DT @RT(4)BOOL @RT(0) @T @T @BASIC 0 @F
@F @F
@T
@BEG_Attrib
3 @RT(0) @RT(0) @RT(0)
@END_Attrib
1 0 @F @F @F @F

@Var @RT(9)miEntries @RT(0) @T @F @DT @RT(4)DINT @RT(0) @T @T @BASIC 0 @F
@F @F
@T
@BEG_Attrib
3 @RT(0) @RT(0) @RT(0)
@END_Attrib
1 0 @F @F @F @F

@Var @RT(12)fbDebugTrace @RT(0) @T @T @DERIVED 0 @F @RT(12)FBDebugTrace @F
@T
@BEG_Attrib
3 @RT(0) @RT(0) @RT(0)
@END_Attrib
1 0 @F @F @F @F

@END_Dcl

@END_Export

@BEG_Body

2

@BEG_Export

@BEG_Algo
@EVENT_ALGORITHM @RT(17)evaAlarmMotorLock @STRUCTURED_TEXT
@RT(0) @RT(16)evAlarmMotorLock @RT(9)EV_Task_3 @F @F
@END_Algo

@BEG_Dcl
@RT(16)DclTreeContainer
2
@Var @RT(20)evAlarmMotorLockData @RT(0) @T @T @DERIVED 0 @F @RT(16)ALARM_EVENT_DATA @F
@T
@BEG_Attrib
3 @RT(0) @RT(0) @RT(0)
@END_Attrib
1 1 @F @F @F @F

@Var @RT(16)ElementMotorLock @RT(0) @T @T @DERIVED 0 @T @T @DT @RT(18)tsElementMotorLock @RT(0) @T @T @UNKNOWN 0 @F
@F @F
@T
@BEG_Attrib
3 @RT(0) @RT(0) @RT(0)
@END_Attrib
1 0 @F @F @F @F

@END_Dcl

@END_Export

@BEG_Export

@BEG_Algo
@EVENT_ALGORITHM @RT(20)evaAlarmMotorRelease @STRUCTURED_TEXT
@RT(0) @RT(19)evAlarmMotorRelease @RT(9)EV_Task_3 @F @F
@END_Algo

@BEG_Dcl
@RT(16)DclTreeContainer
2
@Var @RT(23)evAlarmMotorReleaseData @RT(0) @T @T @DERIVED 0 @T @T @DT @RT(16)ALARM_EVENT_DATA @RT(0) @T @T @UNKNOWN 0 @F
@F @F
@T
@BEG_Attrib
3 @RT(0) @RT(0) @RT(0)
@END_Attrib
1 1 @F @F @F @F

@Var @RT(19)ElementMotorRelease @RT(0) @T @T @DERIVED 0 @T @T @DT @RT(18)tsElementMotorLock @RT(0) @T @T @UNKNOWN 0 @F
@F @F
@T
@BEG_Attrib
3 @RT(0) @RT(0) @RT(0)
@END_Attrib
1 0 @F @F @F @F

@END_Dcl

@END_Export

@BEG_Body
@TL(35)
IF NOT mbInitDone THEN
    abMotorLockList.aInit();
    mbInitDone := TRUE;
END_IF;

IF sv_TraceLevel.bLockUnlock THEN
   fbDebugTrace(CONCAT('motor locked   by alarm ', GET_ALARM_NAME(evAlarmMotorLockData.NAME)));
END_IF;

//search if entry already exists
ElementMotorLock.SearchData.Alarm := evAlarmMotorLockData.NAME;
ElementMotorLock.SearchData.SubID1 := evAlarmMotorLockData.SUBID1;
ElementMotorLock.SearchData.SubID2 := evAlarmMotorLockData.SUBID2;
ElementMotorLock.SearchData.SubID3 := evAlarmMotorLockData.SUBID3;
ElementMotorLock.SearchData.SubID4 := evAlarmMotorLockData.SUBID4;

abMotorLockList.aSearch(SearchData := ElementMotorLock.SearchData);

IF NOT abMotorLockList.aSearch.bFound THEN
    //add entry
    ElementMotorLock.ElementData.Alarm := evAlarmMotorLockData.NAME;
    ElementMotorLock.ElementData.SubID1 := evAlarmMotorLockData.SUBID1;
    ElementMotorLock.ElementData.SubID2 := evAlarmMotorLockData.SUBID2;
    ElementMotorLock.ElementData.SubID3 := evAlarmMotorLockData.SUBID3;
    ElementMotorLock.ElementData.SubID4 := evAlarmMotorLockData.SUBID4;
    abMotorLockList.aAdd(Element := ElementMotorLock);
END_IF;

//get number of elements
miEntries := abMotorLockList.aGetElementCount();
IF miEntries > 0 THEN
    //one or more entries in the list -> release motor
    sv_bMotorLocked := TRUE;
END_IF;

@END_Body

@@@BEG_Comment@@@
@TL(0)

@@@END_Comment@@@

@BEG_Body
@TL(30)
IF NOT mbInitDone THEN
    abMotorLockList.aInit();
    mbInitDone := TRUE;
END_IF;

IF sv_TraceLevel.bLockUnlock THEN
   fbDebugTrace(CONCAT('motor unlocked by alarm ', GET_ALARM_NAME(evAlarmMotorReleaseData.NAME)));
END_IF;

//search if entry already exists
ElementMotorRelease.SearchData.Alarm := evAlarmMotorReleaseData.NAME;
ElementMotorRelease.SearchData.SubID1 := evAlarmMotorReleaseData.SUBID1;
ElementMotorRelease.SearchData.SubID2 := evAlarmMotorReleaseData.SUBID2;
ElementMotorRelease.SearchData.SubID3 := evAlarmMotorReleaseData.SUBID3;
ElementMotorRelease.SearchData.SubID4 := evAlarmMotorReleaseData.SUBID4;

abMotorLockList.aSearch(SearchData := ElementMotorRelease.SearchData);

IF abMotorLockList.aSearch.bFound THEN
    //remove entry
    abMotorLockList.aRemove(SearchData := ElementMotorRelease.SearchData);
END_IF;

//get number of elements
miEntries := abMotorLockList.aGetElementCount();
IF miEntries = 0 THEN
    //no lock entries left -> release motor
    sv_bMotorLocked := FALSE;
END_IF;

@END_Body

@@@BEG_Comment@@@
@TL(0)

@@@END_Comment@@@
@END_Body

@END_Contents

(* ---- ABMovementHistory.pu ---- *)
(*
@h    ! WARNING !
@h    The Kemro K2 system (including software) only meets category B according to EN 954-1,
@h    thus it is not intended for usage in safety-relevant control applications in the field
@h    of personal safety (e.g. emergency stop).
@h    To implement potentially necessary safety-relevant control tasks, always use additional
@h    external safety devices that are intended for the particular purpose, and meet the necessary
@h    functional safety.
@h    For further information see EN 954-1 (EN ISO 13849-1) and/or the K2-x00 user manual, chapter
@h    "CE conformity, directives and standards".

This AB saves executed movements a list (sv_MovementHistory).
Only movements in HA or FA are saved in this list.
If operation mode changes to manual or setup or if the shotcounter is increased the list is resetted.
*)

IMPORT_OVER_LISTFILE
 cMoveNone
, cMinMoveIdent
, tsMovementHistory
, tnOperationMode
, tsMoveCtrl

END_IMPORT

ALGORITHM_BLOCK ABMovementHistory #DUMMY_EDIT_BLOCK

SYSTEM_VAR
 sv_MovementHistory : tsMovementHistory;
 sv_iShotCounterAct : DINT;
 sv_OperationMode : tnOperationMode;
 sv_bStepBwdActive : BOOL (* TRUE: stepping bwd is active *);
END_VAR

SYSTEM_OBJECT
 PU_Task_3 : TASK;
 PU_Task_7 : TASK;
END_OBJECT

VAR_EXTERNAL
 g_MoveCtrl : tsMoveCtrl;
END_VAR

ALGORITHM aResetList

VAR_TEMP
 i : DINT;
END_VAR
#BEGIN_EDIT_BLOCK
(**************************************** WARNING ********************************************
 *** The KEBA Kemro K2 System including software is not intended for safety control tasks! ***
 ***                       For further information see Comment tab!                        ***
 *********************************************************************************************)

FOR i := 1 TO sv_MovementHistory.iActCount DO
   sv_MovementHistory.Data[i].MoveDir := cMoveNone;
   sv_MovementHistory.Data[i].MoveId := cMinMoveIdent;
   sv_MovementHistory.Data[i].iCount := 0;
END_FOR;

sv_MovementHistory.iActCount := 0;

;#END_EDIT_BLOCK END_ALGORITHM

ALGORITHM aAddMovement

VAR_INPUT
 MoveId : DINT;
 MoveDir : DINT;
 iCount : DINT;
END_VAR

VAR
 bEqual : BOOL;
END_VAR
#BEGIN_EDIT_BLOCK
(**************************************** WARNING ********************************************
 *** The KEBA Kemro K2 System including software is not intended for safety control tasks! ***
 ***                       For further information see Comment tab!                        ***
 *********************************************************************************************)

IF (sv_MovementHistory.iActCount < cMovementHistoryLength) THEN

   //only add if it is different from the last entry
   IF sv_MovementHistory.iActCount > 0 THEN
      bEqual := (sv_MovementHistory.Data[sv_MovementHistory.iActCount].MoveDir = MoveDir) AND
             (sv_MovementHistory.Data[sv_MovementHistory.iActCount].MoveId = MoveId) AND
             (sv_MovementHistory.Data[sv_MovementHistory.iActCount].iCount = iCount);
   ELSE
      bEqual := FALSE;
   END_IF;

   IF NOT bEqual THEN
      sv_MovementHistory.iActCount := sv_MovementHistory.iActCount + 1;
      sv_MovementHistory.Data[sv_MovementHistory.iActCount].MoveDir := MoveDir;
      sv_MovementHistory.Data[sv_MovementHistory.iActCount].MoveId := MoveId;
      sv_MovementHistory.Data[sv_MovementHistory.iActCount].iCount := iCount;
   END_IF;

END_IF;

;#END_EDIT_BLOCK END_ALGORITHM

ALGORITHM aRemoveMovement

#BEGIN_EDIT_BLOCK
(**************************************** WARNING ********************************************
 *** The KEBA Kemro K2 System including software is not intended for safety control tasks! ***
 ***                       For further information see Comment tab!                        ***
 *********************************************************************************************)

IF sv_MovementHistory.iActCount > 0 THEN
   sv_MovementHistory.Data[sv_MovementHistory.iActCount].MoveDir := cMoveNone;
   sv_MovementHistory.Data[sv_MovementHistory.iActCount].MoveId := cMinMoveIdent;
   sv_MovementHistory.Data[sv_MovementHistory.iActCount].iCount := 0;
   sv_MovementHistory.iActCount := (sv_MovementHistory.iActCount - 1);
END_IF;

;#END_EDIT_BLOCK END_ALGORITHM

POSTUPDATE_ALGORITHM pShotCounter ON PU_Task_3 WITH sv_iShotCounterAct

#BEGIN_EDIT_BLOCK
(**************************************** WARNING ********************************************
 *** The KEBA Kemro K2 System including software is not intended for safety control tasks! ***
 ***                       For further information see Comment tab!                        ***
 *********************************************************************************************)

aResetList();

;#END_EDIT_BLOCK END_ALGORITHM

POSTUPDATE_ALGORITHM pOpMode ON PU_Task_7 WITH sv_OperationMode

#BEGIN_EDIT_BLOCK
(**************************************** WARNING ********************************************
 *** The KEBA Kemro K2 System including software is not intended for safety control tasks! ***
 ***                       For further information see Comment tab!                        ***
 *********************************************************************************************)

IF sv_OperationMode < nHalfAutomatic THEN
   aResetList();
END_IF;

;#END_EDIT_BLOCK END_ALGORITHM

ALGORITHM aUpdate

#BEGIN_EDIT_BLOCK
(**************************************** WARNING ********************************************
 *** The KEBA Kemro K2 System including software is not intended for safety control tasks! ***
 ***                       For further information see Comment tab!                        ***
 *********************************************************************************************)

//only add movements which finish successfully (without bStop) in HA an FA mode
IF (sv_OperationMode >= nHalfAutomatic) THEN //AND (NOT g_MoveCtrl.bStop) THEN
   IF sv_bStepBwdActive AND (NOT g_MoveCtrl.bStop) THEN
      aRemoveMovement();
   ELSIF NOT sv_bStepBwdActive THEN
      aAddMovement(MoveId := g_MoveCtrl.pData^.MoveId,
                   MoveDir := g_MoveCtrl.pData^.MoveDir,
                   iCount :=  g_MoveCtrl.iCount);
   END_IF;
END_IF;

;#END_EDIT_BLOCK END_ALGORITHM

END_ALGORITHM_BLOCK

#END_OF_IEC_PART

@Puma @IecEditor 6 138 @Pou 25
@@@BEG_Comment@@@
@h    ! WARNING !
@h    The Kemro K2 system (including software) only meets category B according to EN 954-1,
@h    thus it is not intended for usage in safety-relevant control applications in the field
@h    of personal safety (e.g. emergency stop).
@h    To implement potentially necessary safety-relevant control tasks, always use additional
@h    external safety devices that are intended for the particular purpose, and meet the necessary
@h    functional safety.
@h    For further information see EN 954-1 (EN ISO 13849-1) and/or the K2-x00 user manual, chapter
@h    "CE conformity, directives and standards".

This AB saves executed movements a list (sv_MovementHistory).
Only movements in HA or FA are saved in this list.
If operation mode changes to manual or setup or if the shotcounter is increased the list is resetted.
@@@END_Comment@@@

@BEG_Contents

@BEG_Func
@RT(17)FuncTreeContainer
0
@END_Func

@BEG_Const
@RT(18)ConstTreeContainer
2
@Var @RT(9)cMoveNone @RT(0) @T @F @DT @RT(4)DINT @RT(0) @T @T @BASIC 0 @F
@F @F
@T
@BEG_Attrib
0 @RT(13)cMinMoveIdent @RT(4)None
@END_Attrib
1 1 @F @F @F @F

@Var @RT(13)cMinMoveIdent @RT(0) @T @F @DT @RT(4)DINT @RT(0) @T @T @BASIC 0 @F
@F @F
@T
@BEG_Attrib
0 @RT(1)1 @RT(32)lower limit for MoveId / MoveDir
@END_Attrib
1 1 @F @F @F @F

@END_Const

@BEG_Export

@BEG_Kind
@ALGORITHM_BLOCK @RT(17)ABMovementHistory @STRUCTURED_TEXT
@RT(0) @RT(0) @RT(0)
@END_Kind

@BEG_Dcl
@RT(16)DclTreeContainer
7
@Var @RT(18)sv_MovementHistory @RT(0) @T @T @DERIVED 0 @F @RT(17)tsMovementHistory @F
@T
@BEG_Attrib
3 @RT(0) @RT(0) @RT(0)
@END_Attrib
1 8 @F @F @F @F

@Var @RT(9)PU_Task_3 @RT(0) @T @T @RENAMED 0 @T @T @DT @RT(4)TASK @RT(0) @T @T @BASIC 0 @F
@F @F
@T
@BEG_Attrib
3 @RT(0) @RT(0) @RT(0)
@END_Attrib
1 7 @F @F @F @F

@Var @RT(18)sv_iShotCounterAct @RT(0) @T @T @RENAMED 0 @T @T @DT @RT(4)DINT @RT(0) @T @T @BASIC 0 @F
@F @F
@T
@BEG_Attrib
3 @RT(0) @RT(0) @RT(0)
@END_Attrib
1 8 @F @F @F @F

@Var @RT(9)PU_Task_7 @RT(0) @T @T @RENAMED 0 @T @T @DT @RT(4)TASK @RT(0) @T @T @BASIC 0 @F
@F @F
@T
@BEG_Attrib
3 @RT(0) @RT(0) @RT(0)
@END_Attrib
1 7 @F @F @F @F

@Var @RT(16)sv_OperationMode @RT(0) @T @T @RENAMED 0 @T @T @DT @RT(15)tnOperationMode @RT(0) @T @T @UNKNOWN 0 @F
@F @F
@T
@BEG_Attrib
3 @RT(0) @RT(0) @RT(0)
@END_Attrib
1 8 @F @F @F @F

@Var @RT(10)g_MoveCtrl @RT(0) @T @T @DERIVED 0 @T @T @DT @RT(10)tsMoveCtrl @RT(0) @T @T @UNKNOWN 0 @F
@F @F
@T
@BEG_Attrib
3 @RT(0) @RT(0) @RT(0)
@END_Attrib
1 6 @F @F @F @F

@Var @RT(17)sv_bStepBwdActive @RT(0) @T @F @DT @RT(4)BOOL @RT(0) @T @T @BASIC 0 @F
@F @F
@T
@BEG_Attrib
3 @RT(0) @RT(28)TRUE: stepping bwd is active @RT(0)
@END_Attrib
1 8 @F @F @F @F

@END_Dcl

@END_Export

@BEG_Body

6

@BEG_Export

@BEG_Algo
@ALGORITHM @RT(10)aResetList @STRUCTURED_TEXT
@RT(0) @RT(0) @RT(0) @F @F
@END_Algo

@BEG_Dcl
@RT(16)DclTreeContainer
1
@Var @RT(1)i @RT(0) @T @F @DT @RT(4)DINT @RT(0) @T @T @BASIC 0 @F
@F @F
@T
@BEG_Attrib
3 @RT(0) @RT(0) @RT(0)
@END_Attrib
1 4 @F @F @F @F

@END_Dcl

@END_Export

@BEG_Export

@BEG_Algo
@ALGORITHM @RT(12)aAddMovement @STRUCTURED_TEXT
@RT(0) @RT(0) @RT(0) @F @F
@END_Algo

@BEG_Dcl
@RT(16)DclTreeContainer
4
@Var @RT(6)MoveId @RT(0) @T @F @DT @RT(4)DINT @RT(0) @T @T @BASIC 0 @F
@F @F
@T
@BEG_Attrib
3 @RT(0) @RT(0) @RT(0)
@END_Attrib
1 1 @F @F @F @F

@Var @RT(7)MoveDir @RT(0) @T @F @DT @RT(4)DINT @RT(0) @T @T @BASIC 0 @F
@F @F
@T
@BEG_Attrib
3 @RT(0) @RT(0) @RT(0)
@END_Attrib
1 1 @F @F @F @F

@Var @RT(6)iCount @RT(0) @T @F @DT @RT(4)DINT @RT(0) @T @T @BASIC 0 @F
@F @F
@T
@BEG_Attrib
3 @RT(0) @RT(0) @RT(0)
@END_Attrib
1 1 @F @F @F @F

@Var @RT(6)bEqual @RT(0) @T @F @DT @RT(4)BOOL @RT(0) @T @T @BASIC 0 @F
@F @F
@T
@BEG_Attrib
3 @RT(0) @RT(0) @RT(0)
@END_Attrib
1 0 @F @F @F @F

@END_Dcl

@END_Export

@BEG_Export

@BEG_Algo
@ALGORITHM @RT(15)aRemoveMovement @STRUCTURED_TEXT
@RT(0) @RT(0) @RT(0) @F @F
@END_Algo

@BEG_Dcl
@RT(16)DclTreeContainer
0
@END_Dcl

@END_Export

@BEG_Export

@BEG_Algo
@POSTUPDATE_ALGORITHM @RT(12)pShotCounter @STRUCTURED_TEXT
@RT(0) @RT(18)sv_iShotCounterAct @RT(9)PU_Task_3 @F @F
@END_Algo

@BEG_Dcl
@RT(16)DclTreeContainer
0
@END_Dcl

@END_Export

@BEG_Export

@BEG_Algo
@POSTUPDATE_ALGORITHM @RT(7)pOpMode @STRUCTURED_TEXT
@RT(0) @RT(16)sv_OperationMode @RT(9)PU_Task_7 @F @F
@END_Algo

@BEG_Dcl
@RT(16)DclTreeContainer
0
@END_Dcl

@END_Export

@BEG_Export

@BEG_Algo
@ALGORITHM @RT(7)aUpdate @STRUCTURED_TEXT
@RT(0) @RT(0) @RT(0) @F @F
@END_Algo

@BEG_Dcl
@RT(16)DclTreeContainer
0
@END_Dcl

@END_Export

@BEG_Body
@TL(13)
(**************************************** WARNING ********************************************
 *** The KEBA Kemro K2 System including software is not intended for safety control tasks! ***
 ***                       For further information see Comment tab!                        ***
 *********************************************************************************************)

FOR i := 1 TO sv_MovementHistory.iActCount DO
   sv_MovementHistory.Data[i].MoveDir := cMoveNone;
   sv_MovementHistory.Data[i].MoveId := cMinMoveIdent;
   sv_MovementHistory.Data[i].iCount := 0;
END_FOR;

sv_MovementHistory.iActCount := 0;

@END_Body

@@@BEG_Comment@@@
@TL(0)

@@@END_Comment@@@

@BEG_Body
@TL(25)
(**************************************** WARNING ********************************************
 *** The KEBA Kemro K2 System including software is not intended for safety control tasks! ***
 ***                       For further information see Comment tab!                        ***
 *********************************************************************************************)

IF (sv_MovementHistory.iActCount < cMovementHistoryLength) THEN

   //only add if it is different from the last entry
   IF sv_MovementHistory.iActCount > 0 THEN
      bEqual := (sv_MovementHistory.Data[sv_MovementHistory.iActCount].MoveDir = MoveDir) AND
             (sv_MovementHistory.Data[sv_MovementHistory.iActCount].MoveId = MoveId) AND
             (sv_MovementHistory.Data[sv_MovementHistory.iActCount].iCount = iCount);
   ELSE
      bEqual := FALSE;
   END_IF;

   IF NOT bEqual THEN
      sv_MovementHistory.iActCount := sv_MovementHistory.iActCount + 1;
      sv_MovementHistory.Data[sv_MovementHistory.iActCount].MoveDir := MoveDir;
      sv_MovementHistory.Data[sv_MovementHistory.iActCount].MoveId := MoveId;
      sv_MovementHistory.Data[sv_MovementHistory.iActCount].iCount := iCount;
   END_IF;

END_IF;

@END_Body

@@@BEG_Comment@@@
@TL(0)

@@@END_Comment@@@

@BEG_Body
@TL(14)
(**************************************** WARNING ********************************************
 *** The KEBA Kemro K2 System including software is not intended for safety control tasks! ***
 ***                       For further information see Comment tab!                        ***
 *********************************************************************************************)

IF sv_MovementHistory.iActCount > 0 THEN
   sv_MovementHistory.Data[sv_MovementHistory.iActCount].MoveDir := cMoveNone;
   sv_MovementHistory.Data[sv_MovementHistory.iActCount].MoveId := cMinMoveIdent;
   sv_MovementHistory.Data[sv_MovementHistory.iActCount].iCount := 0;
   sv_MovementHistory.iActCount := (sv_MovementHistory.iActCount - 1);
END_IF;

@END_Body

@@@BEG_Comment@@@
@TL(0)

@@@END_Comment@@@

@BEG_Body
@TL(7)
(**************************************** WARNING ********************************************
 *** The KEBA Kemro K2 System including software is not intended for safety control tasks! ***
 ***                       For further information see Comment tab!                        ***
 *********************************************************************************************)

aResetList();

@END_Body

@@@BEG_Comment@@@
@TL(0)

@@@END_Comment@@@

@BEG_Body
@TL(9)
(**************************************** WARNING ********************************************
 *** The KEBA Kemro K2 System including software is not intended for safety control tasks! ***
 ***                       For further information see Comment tab!                        ***
 *********************************************************************************************)

IF sv_OperationMode < nHalfAutomatic THEN
   aResetList();
END_IF;

@END_Body

@@@BEG_Comment@@@
@TL(0)

@@@END_Comment@@@

@BEG_Body
@TL(16)
(**************************************** WARNING ********************************************
 *** The KEBA Kemro K2 System including software is not intended for safety control tasks! ***
 ***                       For further information see Comment tab!                        ***
 *********************************************************************************************)

//only add movements which finish successfully (without bStop) in HA an FA mode
IF (sv_OperationMode >= nHalfAutomatic) THEN //AND (NOT g_MoveCtrl.bStop) THEN
   IF sv_bStepBwdActive AND (NOT g_MoveCtrl.bStop) THEN
      aRemoveMovement();
   ELSIF NOT sv_bStepBwdActive THEN
      aAddMovement(MoveId := g_MoveCtrl.pData^.MoveId,
                   MoveDir := g_MoveCtrl.pData^.MoveDir,
                   iCount :=  g_MoveCtrl.iCount);
   END_IF;
END_IF;

@END_Body

@@@BEG_Comment@@@
@TL(0)

@@@END_Comment@@@
@END_Body

@END_Contents

(* ---- ABMovementRegister.pu ---- *)
(*
@h    ! WARNING !
@h    The Kemro K2 system (including software) only meets category B according to EN 954-1,
@h    thus it is not intended for usage in safety-relevant control applications in the field
@h    of personal safety (e.g. emergency stop).
@h    To implement potentially necessary safety-relevant control tasks, always use additional
@h    external safety devices that are intended for the particular purpose, and meet the necessary
@h    functional safety.
@h    For further information see EN 954-1 (EN ISO 13849-1) and/or the K2-x00 user manual, chapter
@h    "CE conformity, directives and standards".

Register a movement in the system.
*)

IMPORT_OVER_LISTFILE
 SET_ALARM
, START_PROCESS_ALGORITHM
, ASSERT
, tevMovementRegister
, tsDeviceId
, tyMoveDataArray
, tevMovementRegisterData
, tsMoveData
, ABRegisterDelay

END_IMPORT

ALGORITHM_BLOCK ABMovementRegister #DUMMY_EDIT_BLOCK

SYSTEM_VAR
 sv_DeviceId : tsDeviceId;
 sv_bDeviceReady : BOOL;
 sv_NumberOfMovements : DINT;
 sv_Movements : tyMoveDataArray;
 sv_bAllPUTasksExecuted : BOOL;
END_VAR

SYSTEM_OBJECT
 Task10ms : TASK;
 erNoSvMove : ALARM;
 erMaxMovementsExeeded : ALARM;
 erNoSvDeviceReady : ALARM;
 erAssert : ALARM;
 evMovementRegister : tevMovementRegister;
END_OBJECT

VAR
 evMovementRegisterData : tevMovementRegisterData;
 mpMovementData : REFTO tsMoveData;
END_VAR

(*
Register the movement identified by pMovementData.
For each movement a separate ABMovementRegister block is necessary.
It is not allowed to call aRegister more than once.
*)

ALGORITHM aRegister

VAR_INPUT
 pMovementData : REFTO tsMoveData;
END_VAR

VAR
 bAlreadyCalled : BOOL;
 b : BOOL;
 dummy : DINT;
END_VAR
#BEGIN_EDIT_BLOCK
(**************************************** WARNING ********************************************
 *** The KEBA Kemro K2 System including software is not intended for safety control tasks! ***
 ***                       For further information see Comment tab!                        ***
 *********************************************************************************************)

IF bAlreadyCalled THEN
   //it is not allowed to call aRegister more than once
   dummy := Print('ABMovementRegister.aRegister called multiple times.$nUse a separate ABMovementRegister for each movement to register!');
   b := ASSERT(FALSE, erAssert);
   RETURN;
END_IF;

mpMovementData := pMovementData;

//arm registration
evMovementRegisterData.DeviceId :=  sv_DeviceId;
evMovementRegisterData.Mode := nMoveRegModeArm;
SET_EVENT(evMovementRegister, evMovementRegisterData);

START_PROCESS_ALGORITHM(paDelay);
bAlreadyCalled := TRUE;

;#END_EDIT_BLOCK END_ALGORITHM

(*
@i for registering a movment 2 evMovemnetRegister is sent twice
@i the first one with the mode nMoveRegModeArm, then a delaytime is waited and the event is sent again
@i with the mode nMoveRegModeFire.
@i this is necessary to notice the start and the end of the movmentregistration.

*)

PROCESS_ALGORITHM paDelay ON Task10ms

VAR
 abRegisterDelay : ABRegisterDelay;
END_VAR

(* IecGraph-Code *)

(* init step *)
INITIAL_STEP INIT: (*sv_bInitStart is TRUE and all relevant PU - tasks and EV - tasks are
executed at least one time*)
END_STEP

(* steps *)
STEP WAIT:
Action1 (P);
END_STEP

ACTION Action1: #BEGIN_EDIT_BLOCK
//get registration delaytime
abRegisterDelay.aGet();

;#END_EDIT_BLOCK END_ACTION (*Action1*)
STEP REG:
aRegisterMovement (P);
END_STEP

ACTION aRegisterMovement: #BEGIN_EDIT_BLOCK
START_PROCESS_ALGORITHM(paSetRegisterEventFire);
STOP_PROCESS_ALGORITHM();

;#END_EDIT_BLOCK END_ACTION (*aRegisterMovement*)

(* transitions *)
TRANSITION Trans4 (* Trans4 *) FROM INIT TO WAIT :=  #BEGIN_EDIT_BLOCK
sv_bAllPUTasksExecuted

;#END_EDIT_BLOCK
END_TRANSITION

TRANSITION Trans2 (* Trans2 *) FROM WAIT TO REG :=  #BEGIN_EDIT_BLOCK
WAIT.T >= abRegisterDelay.aGet.Time
;#END_EDIT_BLOCK
END_TRANSITION

(* end IecGraph-Code *)
(* sfc-code *)
(* end sfc-code *)

END_ALGORITHM

PROCESS_ALGORITHM paSetRegisterEventFire ON Task10ms

#BEGIN_EDIT_BLOCK
(**************************************** WARNING ********************************************
 *** The KEBA Kemro K2 System including software is not intended for safety control tasks! ***
 ***                       For further information see Comment tab!                        ***
 *********************************************************************************************)

IF CHECK_REF(mpMovementData^) THEN
   IF  IS_LINKED(sv_bDeviceReady) THEN
      IF sv_NumberOfMovements < cMaxDeviceMovements THEN
         // add reference of sv_MoveXxx to the movementarray
         sv_NumberOfMovements := sv_NumberOfMovements + 1;
         sv_Movements[sv_NumberOfMovements] := mpMovementData;

         //sending registration-event to CentralCoordination
         evMovementRegisterData.sFuName := GET_MY_FU_NAME();
         evMovementRegisterData.Mode := nMoveRegModeFire;
         evMovementRegisterData.DeviceId :=  sv_DeviceId;
         evMovementRegisterData.pbDeviceReady := @sv_bDeviceReady;
         evMovementRegisterData.pMovementData := mpMovementData;
         SET_EVENT(evMovementRegister, evMovementRegisterData);
      ELSE
         // too much movements registered
         SET_ALARM(Name := erMaxMovementsExeeded,
                  SubID1 := sv_DeviceId.CompId,
                  SubID2 := sv_DeviceId.IndexId,
                  SubID3 := cMaxDeviceMovements);
      END_IF;
   ELSE
      // sv_bDeviceReady missing
      SET_ALARM(Name := erNoSvDeviceReady,
                SubID1 := sv_DeviceId.CompId);
   END_IF;
ELSE
   // reference of sv_MoveXxx not valid
   SET_ALARM(Name := erNoSvMove,
            SubID1 := sv_DeviceId.CompId);
END_IF;

STOP_PROCESS_ALGORITHM();

;#END_EDIT_BLOCK END_ALGORITHM

END_ALGORITHM_BLOCK

#END_OF_IEC_PART

@Puma @IecEditor 6 97 @Pou 25
@@@BEG_Comment@@@
@h    ! WARNING !
@h    The Kemro K2 system (including software) only meets category B according to EN 954-1,
@h    thus it is not intended for usage in safety-relevant control applications in the field
@h    of personal safety (e.g. emergency stop).
@h    To implement potentially necessary safety-relevant control tasks, always use additional
@h    external safety devices that are intended for the particular purpose, and meet the necessary
@h    functional safety.
@h    For further information see EN 954-1 (EN ISO 13849-1) and/or the K2-x00 user manual, chapter
@h    "CE conformity, directives and standards".

Register a movement in the system.
@@@END_Comment@@@

@BEG_Contents

@BEG_Func
@RT(17)FuncTreeContainer
3
@Var @RT(9)SET_ALARM @RT(0) @T @T @DERIVED 0 @F @RT(23)KEBA_STANDARD_PROCEDURE @F
@T
@BEG_Attrib
0 @RT(0) @RT(0)
@END_Attrib
1 1 @F @F @F @F

@Var @RT(23)START_PROCESS_ALGORITHM @RT(0) @T @T @DERIVED 0 @F @RT(23)KEBA_STANDARD_PROCEDURE @F
@T
@BEG_Attrib
0 @RT(0) @RT(0)
@END_Attrib
1 1 @F @F @F @F

@Var @RT(6)ASSERT @RT(0) @T @T @DERIVED 0 @F @RT(8)FUNCTION @F
@T
@BEG_Attrib
0 @RT(0) @RT(0)
@END_Attrib
1 1 @F @F @F @F

@END_Func

@BEG_Const
@RT(18)ConstTreeContainer
0
@END_Const

@BEG_Export

@BEG_Kind
@ALGORITHM_BLOCK @RT(18)ABMovementRegister @STRUCTURED_TEXT
@RT(0) @RT(0) @RT(0)
@END_Kind

@BEG_Dcl
@RT(16)DclTreeContainer
13
@Var @RT(8)Task10ms @RT(0) @T @T @RENAMED 0 @T @T @DT @RT(4)TASK @RT(0) @T @T @BASIC 0 @F
@F @F
@T
@BEG_Attrib
3 @RT(0) @RT(0) @RT(0)
@END_Attrib
1 7 @F @F @F @F

@Var @RT(10)erNoSvMove @RT(0) @T @F @DT @RT(5)ALARM @RT(0) @T @T @BASIC 0 @F
@F @F
@T
@BEG_Attrib
3 @RT(0) @RT(0) @RT(0)
@END_Attrib
1 7 @F @F @F @F

@Var @RT(21)erMaxMovementsExeeded @RT(0) @T @F @DT @RT(5)ALARM @RT(0) @T @T @BASIC 0 @F
@F @F
@T
@BEG_Attrib
3 @RT(0) @RT(0) @RT(0)
@END_Attrib
1 7 @F @F @F @F

@Var @RT(17)erNoSvDeviceReady @RT(0) @T @F @DT @RT(5)ALARM @RT(0) @T @T @BASIC 0 @F
@F @F
@T
@BEG_Attrib
3 @RT(0) @RT(0) @RT(0)
@END_Attrib
1 7 @F @F @F @F

@Var @RT(8)erAssert @RT(0) @T @T @RENAMED 0 @T @T @DT @RT(5)ALARM @RT(0) @T @T @BASIC 0 @F
@F @F
@T
@BEG_Attrib
3 @RT(0) @RT(0) @RT(0)
@END_Attrib
1 7 @F @F @F @F

@Var @RT(18)evMovementRegister @RT(0) @T @T @DERIVED 0 @T @T @DT @RT(19)tevMovementRegister @RT(0) @T @T @UNKNOWN 0 @F
@F @F
@T
@BEG_Attrib
3 @RT(0) @RT(0) @RT(0)
@END_Attrib
1 7 @F @F @F @F

@Var @RT(11)sv_DeviceId @RT(0) @T @T @DERIVED 0 @T @T @DT @RT(10)tsDeviceId @RT(0) @T @T @UNKNOWN 0 @F
@F @F
@T
@BEG_Attrib
3 @RT(0) @RT(0) @RT(0)
@END_Attrib
1 8 @F @F @F @F

@Var @RT(15)sv_bDeviceReady @RT(0) @T @F @DT @RT(4)BOOL @RT(0) @T @T @BASIC 0 @F
@F @F
@T
@BEG_Attrib
3 @RT(0) @RT(0) @RT(0)
@END_Attrib
1 8 @F @F @F @F

@Var @RT(20)sv_NumberOfMovements @RT(0) @T @F @DT @RT(4)DINT @RT(0) @T @T @BASIC 0 @F
@F @F
@T
@BEG_Attrib
3 @RT(0) @RT(0) @RT(0)
@END_Attrib
1 8 @F @F @F @F

@Var @RT(12)sv_Movements @RT(0) @T @T @DERIVED 0 @T @T @DT @RT(15)tyMoveDataArray @RT(0) @T @T @UNKNOWN 0 @F
@F @F
@T
@BEG_Attrib
3 @RT(0) @RT(0) @RT(0)
@END_Attrib
1 8 @F @F @F @F

@Var @RT(22)evMovementRegisterData @RT(0) @T @T @DERIVED 0 @T @T @DT @RT(23)tevMovementRegisterData @RT(0) @T @T @UNKNOWN 0 @F
@F @F
@T
@BEG_Attrib
3 @RT(0) @RT(0) @RT(0)
@END_Attrib
1 0 @F @F @F @F

@Var @RT(14)mpMovementData @RT(0) @T @T @REFTO 0 @F @DERIVED 0 @T @T @DT @RT(10)tsMoveData @RT(0) @T @T @UNKNOWN 0 @F
@F @F
@T
@BEG_Attrib
3 @RT(0) @RT(0) @RT(0)
@END_Attrib
1 0 @F @F @F @F

@Var @RT(22)sv_bAllPUTasksExecuted @RT(0) @T @F @DT @RT(4)BOOL @RT(0) @T @T @BASIC 0 @F
@F @F
@T
@BEG_Attrib
3 @RT(0) @RT(0) @RT(0)
@END_Attrib
1 8 @F @F @F @F

@END_Dcl

@END_Export

@BEG_Body

3

@BEG_Export

@BEG_Algo
@ALGORITHM @RT(9)aRegister @STRUCTURED_TEXT
@RT(0) @RT(0) @RT(0) @F @F
@END_Algo

@BEG_Dcl
@RT(16)DclTreeContainer
4
@Var @RT(13)pMovementData @RT(0) @T @T @REFTO 0 @F @DERIVED 0 @T @T @DT @RT(10)tsMoveData @RT(0) @T @T @UNKNOWN 0 @F
@F @F
@T
@BEG_Attrib
3 @RT(0) @RT(0) @RT(0)
@END_Attrib
1 1 @F @F @F @F

@Var @RT(14)bAlreadyCalled @RT(0) @T @F @DT @RT(4)BOOL @RT(0) @T @T @BASIC 0 @F
@F @F
@T
@BEG_Attrib
3 @RT(0) @RT(0) @RT(0)
@END_Attrib
1 0 @F @F @F @F

@Var @RT(1)b @RT(0) @T @F @DT @RT(4)BOOL @RT(0) @T @T @BASIC 0 @F
@F @F
@T
@BEG_Attrib
3 @RT(0) @RT(0) @RT(0)
@END_Attrib
1 0 @F @F @F @F

@Var @RT(5)dummy @RT(0) @T @F @DT @RT(4)DINT @RT(0) @T @T @BASIC 0 @F
@F @F
@T
@BEG_Attrib
3 @RT(0) @RT(0) @RT(0)
@END_Attrib
1 0 @F @F @F @F

@END_Dcl

@END_Export

@BEG_Export

@BEG_Algo
@PROCESS_ALGORITHM @RT(7)paDelay @SEQUENTIAL_FLOW_CHART
@RT(0) @RT(0) @RT(8)Task10ms @F @F
@END_Algo

@BEG_Dcl
@RT(16)DclTreeContainer
1
@Var @RT(15)abRegisterDelay @RT(0) @T @T @DERIVED 0 @T @T @DT @RT(15)ABRegisterDelay @RT(0) @T @T @UNKNOWN 0 @F
@F @F
@T
@BEG_Attrib
3 @RT(0) @RT(0) @RT(0)
@END_Attrib
1 0 @F @F @F @F

@END_Dcl

@END_Export

@BEG_Export

@BEG_Algo
@PROCESS_ALGORITHM @RT(22)paSetRegisterEventFire @STRUCTURED_TEXT
@RT(0) @RT(0) @RT(8)Task10ms @F @F
@END_Algo

@BEG_Dcl
@RT(16)DclTreeContainer
0
@END_Dcl

@END_Export

@BEG_Body
@TL(22)
(**************************************** WARNING ********************************************
 *** The KEBA Kemro K2 System including software is not intended for safety control tasks! ***
 ***                       For further information see Comment tab!                        ***
 *********************************************************************************************)

IF bAlreadyCalled THEN
   //it is not allowed to call aRegister more than once
   dummy := Print('ABMovementRegister.aRegister called multiple times.$nUse a separate ABMovementRegister for each movement to register!');
   b := ASSERT(FALSE, erAssert);
   RETURN;
END_IF;

mpMovementData := pMovementData;

//arm registration
evMovementRegisterData.DeviceId :=  sv_DeviceId;
evMovementRegisterData.Mode := nMoveRegModeArm;
SET_EVENT(evMovementRegister, evMovementRegisterData);

START_PROCESS_ALGORITHM(paDelay);
bAlreadyCalled := TRUE;

@END_Body

@@@BEG_Comment@@@
@TL(3)
Register the movement identified by pMovementData.
For each movement a separate ABMovementRegister block is necessary.
It is not allowed to call aRegister more than once.
@@@END_Comment@@@

@BEG_SfcBody
8 6 5

@BEG_SfcData 2
@StepSeq @RT(4)sseq @F 5
@Step @RT(4)INIT @F @T @F @F @RT(0) @T @TL(2)
sv_bInitStart is TRUE and all relevant PU - tasks and EV - tasks are
executed at least one time

@AcbCont @RT(7)unnamed @F 0

@Trans @RT(6)Trans4 @F @T @F @F @T @T @TL(3)
sv_bAllPUTasksExecuted

@RT(6)Trans4 @F
@Step @RT(4)WAIT @F @F @F @F @RT(0) @F
@AcbCont @RT(7)unnamed @F 1
@Acb @RT(7)Action1 @F @T @RT(1)P @RT(0) @F @F @T @TL(4)
//get registration delaytime
abRegisterDelay.aGet();

@F

@Trans @RT(6)Trans2 @F @T @F @F @T @T @TL(2)
WAIT.T >= abRegisterDelay.aGet.Time

@RT(6)Trans2 @F
@Step @RT(3)REG @F @F @F @F @RT(0) @F
@AcbCont @RT(7)unnamed @F 1
@Acb @RT(17)aRegisterMovement @F @T @RT(1)P @RT(0) @F @F @T @TL(3)
START_PROCESS_ALGORITHM(paSetRegisterEventFire);
STOP_PROCESS_ALGORITHM();

@F

@END_SfcData
@SaActions 0
@SaTrans 0
@SaExits 0
@END_SfcBody

@@@BEG_Comment@@@
@TL(5)
@i for registering a movment 2 evMovemnetRegister is sent twice
@i the first one with the mode nMoveRegModeArm, then a delaytime is waited and the event is sent again
@i with the mode nMoveRegModeFire.
@i this is necessary to notice the start and the end of the movmentregistration.

@@@END_Comment@@@

@BEG_Body
@TL(39)
(**************************************** WARNING ********************************************
 *** The KEBA Kemro K2 System including software is not intended for safety control tasks! ***
 ***                       For further information see Comment tab!                        ***
 *********************************************************************************************)

IF CHECK_REF(mpMovementData^) THEN
   IF  IS_LINKED(sv_bDeviceReady) THEN
      IF sv_NumberOfMovements < cMaxDeviceMovements THEN
         // add reference of sv_MoveXxx to the movementarray
         sv_NumberOfMovements := sv_NumberOfMovements + 1;
         sv_Movements[sv_NumberOfMovements] := mpMovementData;

         //sending registration-event to CentralCoordination
         evMovementRegisterData.sFuName := GET_MY_FU_NAME();
         evMovementRegisterData.Mode := nMoveRegModeFire;
         evMovementRegisterData.DeviceId :=  sv_DeviceId;
         evMovementRegisterData.pbDeviceReady := @sv_bDeviceReady;
         evMovementRegisterData.pMovementData := mpMovementData;
         SET_EVENT(evMovementRegister, evMovementRegisterData);
      ELSE
         // too much movements registered
         SET_ALARM(Name := erMaxMovementsExeeded,
                  SubID1 := sv_DeviceId.CompId,
                  SubID2 := sv_DeviceId.IndexId,
                  SubID3 := cMaxDeviceMovements);
      END_IF;
   ELSE
      // sv_bDeviceReady missing
      SET_ALARM(Name := erNoSvDeviceReady,
                SubID1 := sv_DeviceId.CompId);
   END_IF;
ELSE
   // reference of sv_MoveXxx not valid
   SET_ALARM(Name := erNoSvMove,
            SubID1 := sv_DeviceId.CompId);
END_IF;

STOP_PROCESS_ALGORITHM();

@END_Body

@@@BEG_Comment@@@
@TL(0)

@@@END_Comment@@@
@END_Body

@END_Contents

(* ---- ABMoveTimeLimited.pu ---- *)
(*
start a movement for X seconds
after that time the movement is stopped again
*)

IMPORT_OVER_LISTFILE
 tevStop
, tevStartRequest
, tsDeviceId
, tMoveIdent
, tevStartRequestData
, tevStopData
, TON

END_IMPORT

ALGORITHM_BLOCK ABMoveTimeLimited #DUMMY_EDIT_BLOCK

SYSTEM_OBJECT
 PU_Task_7 : TASK;
 evStop : tevStop;
 evStartRequest : tevStartRequest;
END_OBJECT

VAR
 mbMovementStopped : BOOL (* stop of movement was triggerd before  time elapsed *);
 mDeviceId : tsDeviceId;
 mbRunning : BOOL;
END_VAR

ALGORITHM aMove

VAR_INPUT
 dTime : TIME;
 DeviceId : tsDeviceId;
 MoveDir : tMoveIdent;
 MoveId : tMoveIdent;
END_VAR

VAR_OUTPUT
 bTimeReached : BOOL (* was stopped by time limit *);
 bDone : BOOL (* movement is stopped again *);
END_VAR

VAR
 evStartRequestData : tevStartRequestData;
 evStopData : tevStopData;
 fbTimer : TON;
END_VAR

(* IecGraph-Code *)

(* init step *)
INITIAL_STEP Step1:
aStart (P);
aRunTimer (N);
END_STEP

(* steps *)
STEP Step5:
aStop (N);
END_STEP

STEP Step6:
END_STEP

STEP Step3:
Action2 (N);
END_STEP

ACTION Action2: #BEGIN_EDIT_BLOCK
bDone := TRUE;
mbRunning := FALSE;

;#END_EDIT_BLOCK END_ACTION (*Action2*)

(* transitions *)
TRANSITION Trans1 FROM Step1 TO Step5 :=  #BEGIN_EDIT_BLOCK
fbTimer.Q
;#END_EDIT_BLOCK
END_TRANSITION

GO_ON_TRANSITION Trans5 FROM Step5 TO Step3 :=  #BEGIN_EDIT_BLOCK
TRUE
;#END_EDIT_BLOCK
END_TRANSITION

TRANSITION Trans3 FROM Step1 TO Step6 :=  #BEGIN_EDIT_BLOCK
mbMovementStopped
;#END_EDIT_BLOCK
END_TRANSITION

GO_ON_TRANSITION Trans6 FROM Step6 TO Step3 :=  #BEGIN_EDIT_BLOCK
TRUE
;#END_EDIT_BLOCK
END_TRANSITION

TRANSITION Trans7 FROM Step3 TO Step1 :=  #BEGIN_EDIT_BLOCK
TRUE
;#END_EDIT_BLOCK
END_TRANSITION

(* end IecGraph-Code *)
(* sfc-code *)

(* stand alone actions *)
ACTION aStop: #BEGIN_EDIT_BLOCK

evStopData.DeviceId := DeviceId;
SET_EVENT(evStop, evStopData);

bTimeReached := TRUE;

;#END_EDIT_BLOCK END_ACTION (*aStop*)
ACTION aRunTimer: #BEGIN_EDIT_BLOCK
(**************************************** WARNING ********************************************
 *** The KEBA Kemro K2 System including software is not intended for safety control tasks! ***
 ***                       For further information see Comment tab!                        ***
 *********************************************************************************************)

fbTimer();

;#END_EDIT_BLOCK END_ACTION (*aRunTimer*)
ACTION aStart: #BEGIN_EDIT_BLOCK
(**************************************** WARNING ********************************************
 *** The KEBA Kemro K2 System including software is not intended for safety control tasks! ***
 ***                       For further information see Comment tab!                        ***
 *********************************************************************************************)
fbTimer(IN := FALSE);
fbTimer(IN := TRUE, PT := dTime);

mbMovementStopped := FALSE;
bTimeReached := FALSE;
bDone := FALSE;

//save for later use
mDeviceId := DeviceId;
mbRunning := TRUE;

evStartRequestData.DeviceId := DeviceId;
evStartRequestData.MoveDir := MoveDir;
evStartRequestData.MoveId := MoveId;
SET_EVENT(evStartRequest, evStartRequestData);

;#END_EDIT_BLOCK END_ACTION (*aStart*)
(* end sfc-code *)

END_ALGORITHM

EVENT_ALGORITHM evStopAlgo ON PU_Task_7 WITH evStop

VAR_INPUT
 evStopData : tevStopData;
END_VAR
#BEGIN_EDIT_BLOCK
(**************************************** WARNING ********************************************
 *** The KEBA Kemro K2 System including software is not intended for safety control tasks! ***
 ***                       For further information see Comment tab!                        ***
 *********************************************************************************************)

IF evStopData.DeviceId = mDeviceId AND mbRunning THEN
   mbMovementStopped := TRUE;
END_IF;

;#END_EDIT_BLOCK END_ALGORITHM

END_ALGORITHM_BLOCK

#END_OF_IEC_PART

@Puma @IecEditor 6 30 @Pou 25
@@@BEG_Comment@@@
start a movement for X seconds
after that time the movement is stopped again
@@@END_Comment@@@

@BEG_Contents

@BEG_Func
@RT(17)FuncTreeContainer
0
@END_Func

@BEG_Const
@RT(18)ConstTreeContainer
0
@END_Const

@BEG_Export

@BEG_Kind
@ALGORITHM_BLOCK @RT(17)ABMoveTimeLimited @STRUCTURED_TEXT
@RT(0) @RT(0) @RT(0)
@END_Kind

@BEG_Dcl
@RT(16)DclTreeContainer
6
@Var @RT(9)PU_Task_7 @RT(0) @T @T @RENAMED 0 @T @T @DT @RT(4)TASK @RT(0) @T @T @BASIC 0 @F
@F @F
@T
@BEG_Attrib
3 @RT(0) @RT(0) @RT(0)
@END_Attrib
1 7 @F @F @F @F

@Var @RT(17)mbMovementStopped @RT(0) @T @F @DT @RT(4)BOOL @RT(0) @T @T @BASIC 0 @F
@F @F
@T
@BEG_Attrib
3 @RT(0) @RT(50)stop of movement was triggerd before  time elapsed @RT(0)
@END_Attrib
1 0 @F @F @F @F

@Var @RT(6)evStop @RT(0) @T @T @RENAMED 0 @T @T @DT @RT(7)tevStop @RT(0) @T @T @UNKNOWN 0 @F
@F @F
@T
@BEG_Attrib
3 @RT(0) @RT(0) @RT(0)
@END_Attrib
1 7 @F @F @F @F

@Var @RT(14)evStartRequest @RT(0) @T @T @RENAMED 0 @T @T @DT @RT(15)tevStartRequest @RT(0) @T @T @UNKNOWN 0 @F
@F @F
@T
@BEG_Attrib
3 @RT(0) @RT(0) @RT(0)
@END_Attrib
1 7 @F @F @F @F

@Var @RT(9)mDeviceId @RT(0) @T @T @DERIVED 0 @T @T @DT @RT(10)tsDeviceId @RT(0) @T @T @UNKNOWN 0 @F
@F @F
@T
@BEG_Attrib
3 @RT(0) @RT(0) @RT(0)
@END_Attrib
1 0 @F @F @F @F

@Var @RT(9)mbRunning @RT(0) @T @F @DT @RT(4)BOOL @RT(0) @T @T @BASIC 0 @F
@F @F
@T
@BEG_Attrib
3 @RT(0) @RT(0) @RT(0)
@END_Attrib
1 0 @F @F @F @F

@END_Dcl

@END_Export

@BEG_Body

2

@BEG_Export

@BEG_Algo
@ALGORITHM @RT(5)aMove @SEQUENTIAL_FLOW_CHART
@RT(0) @RT(0) @RT(0) @F @F
@END_Algo

@BEG_Dcl
@RT(16)DclTreeContainer
9
@Var @RT(5)dTime @RT(0) @T @F @DT @RT(4)TIME @RT(0) @T @T @BASIC 0 @F
@F @F
@T
@BEG_Attrib
3 @RT(0) @RT(0) @RT(0)
@END_Attrib
1 1 @F @F @F @F

@Var @RT(8)DeviceId @RT(0) @T @T @DERIVED 0 @T @T @DT @RT(10)tsDeviceId @RT(0) @T @T @UNKNOWN 0 @F
@F @F
@T
@BEG_Attrib
3 @RT(0) @RT(0) @RT(0)
@END_Attrib
1 1 @F @F @F @F

@Var @RT(7)MoveDir @RT(0) @T @T @DERIVED 0 @T @T @DT @RT(10)tMoveIdent @RT(0) @T @T @UNKNOWN 0 @F
@F @F
@T
@BEG_Attrib
3 @RT(0) @RT(0) @RT(0)
@END_Attrib
1 1 @F @F @F @F

@Var @RT(6)MoveId @RT(0) @T @T @DERIVED 0 @T @T @DT @RT(10)tMoveIdent @RT(0) @T @T @UNKNOWN 0 @F
@F @F
@T
@BEG_Attrib
3 @RT(0) @RT(0) @RT(0)
@END_Attrib
1 1 @F @F @F @F

@Var @RT(12)bTimeReached @RT(0) @T @F @DT @RT(4)BOOL @RT(0) @T @T @BASIC 0 @F
@F @F
@T
@BEG_Attrib
3 @RT(0) @RT(25)was stopped by time limit @RT(0)
@END_Attrib
1 3 @F @F @F @F

@Var @RT(5)bDone @RT(0) @T @F @DT @RT(4)BOOL @RT(0) @T @T @BASIC 0 @F
@F @F
@T
@BEG_Attrib
3 @RT(0) @RT(25)movement is stopped again @RT(0)
@END_Attrib
1 3 @F @F @F @F

@Var @RT(18)evStartRequestData @RT(0) @T @T @DERIVED 0 @T @T @DT @RT(19)tevStartRequestData @RT(0) @T @T @UNKNOWN 0 @F
@F @F
@T
@BEG_Attrib
3 @RT(0) @RT(0) @RT(0)
@END_Attrib
1 0 @F @F @F @F

@Var @RT(10)evStopData @RT(0) @T @T @DERIVED 0 @T @T @DT @RT(11)tevStopData @RT(0) @T @T @UNKNOWN 0 @F
@F @F
@T
@BEG_Attrib
3 @RT(0) @RT(0) @RT(0)
@END_Attrib
1 0 @F @F @F @F

@Var @RT(7)fbTimer @RT(0) @T @T @DERIVED 0 @T @T @DT @RT(3)TON @RT(0) @T @T @UNKNOWN 0 @F
@F @F
@T
@BEG_Attrib
3 @RT(0) @RT(0) @RT(0)
@END_Attrib
1 0 @F @F @F @F

@END_Dcl

@END_Export

@BEG_Export

@BEG_Algo
@EVENT_ALGORITHM @RT(10)evStopAlgo @STRUCTURED_TEXT
@RT(0) @RT(6)evStop @RT(9)PU_Task_7 @F @F
@END_Algo

@BEG_Dcl
@RT(16)DclTreeContainer
1
@Var @RT(10)evStopData @RT(0) @T @T @DERIVED 0 @T @T @DT @RT(11)tevStopData @RT(0) @T @T @UNKNOWN 0 @F
@F @F
@T
@BEG_Attrib
3 @RT(0) @RT(0) @RT(0)
@END_Attrib
1 1 @F @F @F @F

@END_Dcl

@END_Export

@BEG_SfcBody
3 2 2

@BEG_SfcData 2
@StepSeq @RT(4)sseq @F 1
@Loop @RT(4)loop @F 2
@StepSeq @RT(3)seq @F 3
@Step @RT(5)Step1 @F @T @F @F @RT(0) @F
@AcbCont @RT(7)unnamed @F 2
@Acb @RT(6)aStart @F @F @RT(1)P @RT(0) @F @F @T @F
@Acb @RT(9)aRunTimer @F @F @RT(1)N @RT(0) @F @F @T @F

@AltBranch @RT(3)alt @F 2
@TransSeq @RT(4)tseq @F 3
@Trans @RT(6)Trans1 @F @T @F @F @T @T @TL(2)
fbTimer.Q

@RT(6)Trans1 @F
@Step @RT(5)Step5 @F @F @F @F @RT(0) @F
@AcbCont @RT(7)unnamed @F 1
@Acb @RT(5)aStop @F @F @RT(1)N @RT(0) @F @F @T @F

@Trans @RT(6)Trans5 @F @T @F @F @T @F @TL(2)
TRUE

@RT(6)Trans5 @F

@TransSeq @RT(4)tseq @F 3
@Trans @RT(6)Trans3 @F @T @F @F @T @T @TL(2)
mbMovementStopped

@RT(6)Trans3 @F
@Step @RT(5)Step6 @F @F @F @F @RT(0) @F
@AcbCont @RT(7)unnamed @F 0

@Trans @RT(6)Trans6 @F @T @F @F @T @F @TL(2)
TRUE

@RT(6)Trans6 @F

@Step @RT(5)Step3 @F @F @F @F @RT(0) @F
@AcbCont @RT(7)unnamed @F 1
@Acb @RT(7)Action2 @F @T @RT(1)N @RT(0) @F @F @T @TL(3)
bDone := TRUE;
mbRunning := FALSE;

@F

@Trans @RT(6)Trans7 @F @T @T @T @T @T @TL(2)
TRUE

@RT(6)Trans7 @F

@END_SfcData
@SaActions 3
@SaText @RT(5)aStop 1 @TL(7)

evStopData.DeviceId := DeviceId;
SET_EVENT(evStop, evStopData);

bTimeReached := TRUE;

@SaText @RT(9)aRunTimer 1 @TL(7)
(**************************************** WARNING ********************************************
 *** The KEBA Kemro K2 System including software is not intended for safety control tasks! ***
 ***                       For further information see Comment tab!                        ***
 *********************************************************************************************)

fbTimer();

@SaText @RT(6)aStart 1 @TL(21)
(**************************************** WARNING ********************************************
 *** The KEBA Kemro K2 System including software is not intended for safety control tasks! ***
 ***                       For further information see Comment tab!                        ***
 *********************************************************************************************)
fbTimer(IN := FALSE);
fbTimer(IN := TRUE, PT := dTime);

mbMovementStopped := FALSE;
bTimeReached := FALSE;
bDone := FALSE;

//save for later use
mDeviceId := DeviceId;
mbRunning := TRUE;

evStartRequestData.DeviceId := DeviceId;
evStartRequestData.MoveDir := MoveDir;
evStartRequestData.MoveId := MoveId;
SET_EVENT(evStartRequest, evStartRequestData);

@SaTrans 0
@SaExits 0
@END_SfcBody

@@@BEG_Comment@@@
@TL(0)

@@@END_Comment@@@

@BEG_Body
@TL(10)
(**************************************** WARNING ********************************************
 *** The KEBA Kemro K2 System including software is not intended for safety control tasks! ***
 ***                       For further information see Comment tab!                        ***
 *********************************************************************************************)

IF evStopData.DeviceId = mDeviceId AND mbRunning THEN
   mbMovementStopped := TRUE;
END_IF;

@END_Body

@@@BEG_Comment@@@
@TL(0)

@@@END_Comment@@@
@END_Body

@END_Contents
